			//
			IF _ResultPosition_CAL > 0 THEN 
				// calibration was completed
				// res: CAL rat:23.23 rot:23.23 err:23.23
				_VisionResult := MID(STR:=_VisionResult,LEN:=LEN(_VisionResult)-LEN(_RESPONSE_CAL),POS:=LEN(_RESPONSE_CAL)+1);
				//VisionStateText := CONCAT(VisionStateText, '\n');
				//VisionStateText := CONCAT(VisionStateText, _VisionResult);
				// rat:23.23 rot:23.23 err:23.23
				_ResultPosition := FIND(STR1:=_VisionResult,STR2:='rat:');
				IF _ResultPosition > 0 THEN
					_VisionResult := MID(STR:=_VisionResult,LEN:=LEN(_VisionResult)-LEN('rat:'),POS:=LEN('rat:')+1);
					_SpacePosition := FIND(STR1:=_VisionResult,STR2:=' ');
					_VisionRatio := STRING_TO_REAL(MID(STR:=_VisionResult,LEN:=_SpacePosition-1,POS:=1));
					_VisionResult := MID(STR:=_VisionResult,LEN:=LEN(_VisionResult)-_SpacePosition,POS:=_SpacePosition+1);
				END_IF
				// rot:23.23 err:23.23
				_ResultPosition := FIND(STR1:=_VisionResult,STR2:='rot:');
				IF _ResultPosition > 0 THEN
					_VisionResult := MID(STR:=_VisionResult,LEN:=LEN(_VisionResult)-LEN('rot:'),POS:=LEN('rot:')+1);
					_SpacePosition := FIND(STR1:=_VisionResult,STR2:=' ');
					_VisionRotation := STRING_TO_REAL(MID(STR:=_VisionResult,LEN:=_SpacePosition-1,POS:=1));
					_VisionResult := MID(STR:=_VisionResult,LEN:=LEN(_VisionResult)-_SpacePosition,POS:=_SpacePosition+1);
				END_IF
				// err:23.23
				_ResultPosition := FIND(STR1:=_VisionResult,STR2:='err:');
				IF _ResultPosition > 0 THEN
					_VisionResult := MID(STR:=_VisionResult,LEN:=LEN(_VisionResult)-LEN('err:'),POS:=LEN('err:')+1);
					_SpacePosition := FIND(STR1:=_VisionResult,STR2:=' ');
					_VisionError := STRING_TO_REAL(MID(STR:=_VisionResult,LEN:=_SpacePosition-1,POS:=1));
					_VisionResult := MID(STR:=_VisionResult,LEN:=LEN(_VisionResult)-_SpacePosition,POS:=_SpacePosition+1);
				END_IF
				
			ELSIF _ResultPosition_LOC > 0 THEN 
				// part was located
				// 'res: LOC obj:0 cx:54.66 cy:119.45 a:-12.87 s:0.84 $NLOC obj:1 cx:71.49 cy:100.06 a:10.13 s:0.83 $N'
				_VisionResult := MID(STR:=_VisionResult,LEN:=LEN(_VisionResult)-LEN(_RESPONSE_LOC),POS:=LEN(_RESPONSE_LOC)+1);
				//VisionStateText := CONCAT(VisionStateText, '\n');
				//VisionStateText := CONCAT(VisionStateText, _VisionResult);
				_VisionObjectIndex := 0;
				WHILE FIND(STR1:=_VisionResult,STR2:='obj:') > 0 
					AND _VisionObjectIndex <= _VisionCommandParser.stCommand.Locate.MaxParts 
					AND _VisionObjectIndex + _VisionCommandParser.stCommand.Locate.ResultPosition < GVL.VIS_ARR_END DO
					// 'obj:0 cx:54.66 cy:119.45 a:-12.87 s:0.84 $NLOC obj:1 cx:71.49 cy:100.06 a:10.13 s:0.83 $N'
					// $NLOC obj:1 cx:71.49 cy:100.06 a:10.13 s:0.83 $N'
					_ResultPosition := FIND(STR1:=_VisionResult,STR2:='obj:');
					IF _ResultPosition > 0 THEN
						_PartsCount := _PartsCount + 1;
						_VisionResult := MID(STR:=_VisionResult,LEN:=LEN(_VisionResult)-_ResultPosition-LEN('obj:')+1,POS:=_ResultPosition+LEN('obj:'));
						_SpacePosition := FIND(STR1:=_VisionResult,STR2:=' ');
						_VisionObjectIndex := STRING_TO_UINT(MID(STR:=_VisionResult,LEN:=_SpacePosition-1,POS:=1));
						SUPER^.VisionRegisters[_VisionCommandParser.stCommand.Locate.ResultPosition + _VisionObjectIndex].Comment := CONCAT('obj:', UDINT_TO_STRING(_VisionObjectIndex));
						_VisionResult := MID(STR:=_VisionResult,LEN:=LEN(_VisionResult)-_SpacePosition,POS:=_SpacePosition+1);
					END_IF
					// cx:54.66 cy:119.45 a:-12.87 s:0.84 $NLOC obj:1 cx:71.49 cy:100.06 a:10.13 s:0.83 $N'
					_ResultPosition := FIND(STR1:=_VisionResult,STR2:='cx:');
					IF _ResultPosition > 0 THEN
						_VisionResult := MID(STR:=_VisionResult,LEN:=LEN(_VisionResult)-LEN('cx:'),POS:=LEN('cx:')+1);
						_SpacePosition := FIND(STR1:=_VisionResult,STR2:=' ');
						SUPER^.VisionRegisters[_VisionCommandParser.stCommand.Locate.ResultPosition + _VisionObjectIndex].Position.X := STRING_TO_LREAL(MID(STR:=_VisionResult,LEN:=_SpacePosition-1,POS:=1));
						_VisionResult := MID(STR:=_VisionResult,LEN:=LEN(_VisionResult)-_SpacePosition,POS:=_SpacePosition+1);
					END_IF
					// cy:119.45 a:-12.87 s:0.84 $NLOC obj:1 cx:71.49 cy:100.06 a:10.13 s:0.83 $N'
					_ResultPosition := FIND(STR1:=_VisionResult,STR2:='cy:');
					IF _ResultPosition > 0 THEN
						_VisionResult := MID(STR:=_VisionResult,LEN:=LEN(_VisionResult)-LEN('cy:'),POS:=LEN('cy:')+1);
						_SpacePosition := FIND(STR1:=_VisionResult,STR2:=' ');
						SUPER^.VisionRegisters[_VisionCommandParser.stCommand.Locate.ResultPosition + _VisionObjectIndex].Position.Y := STRING_TO_LREAL(MID(STR:=_VisionResult,LEN:=_SpacePosition-1,POS:=1));
						_VisionResult := MID(STR:=_VisionResult,LEN:=LEN(_VisionResult)-_SpacePosition,POS:=_SpacePosition+1);
					END_IF
					// a:-12.87 s:0.84 $NLOC obj:1 cx:71.49 cy:100.06 a:10.13 s:0.83 $N'
					_ResultPosition := FIND(STR1:=_VisionResult,STR2:='a:');
					IF _ResultPosition > 0 THEN
						_VisionResult := MID(STR:=_VisionResult,LEN:=LEN(_VisionResult)-LEN('a:'),POS:=LEN('a:')+1);
						_SpacePosition := FIND(STR1:=_VisionResult,STR2:=' ');
						SUPER^.VisionRegisters[_VisionCommandParser.stCommand.Locate.ResultPosition + _VisionObjectIndex].Position.A := STRING_TO_LREAL(MID(STR:=_VisionResult,LEN:=_SpacePosition-1,POS:=1));
						_VisionResult := MID(STR:=_VisionResult,LEN:=LEN(_VisionResult)-_SpacePosition,POS:=_SpacePosition+1);
					END_IF
					// s:0.84 $NLOC obj:1 cx:71.49 cy:100.06 a:10.13 s:0.83 $N'
					_ResultPosition := FIND(STR1:=_VisionResult,STR2:='s:');
					IF _ResultPosition > 0 THEN
						_VisionResult := MID(STR:=_VisionResult,LEN:=LEN(_VisionResult)-LEN('s:'),POS:=LEN('s:')+1);
						_SpacePosition := FIND(STR1:=_VisionResult,STR2:=' ');
						SUPER^.VisionRegisters[_VisionCommandParser.stCommand.Locate.ResultPosition + _VisionObjectIndex].Scaling := STRING_TO_REAL(MID(STR:=_VisionResult,LEN:=_SpacePosition-1,POS:=1));
						_VisionResult := MID(STR:=_VisionResult,LEN:=LEN(_VisionResult)-_SpacePosition,POS:=_SpacePosition+1);
					END_IF
					// $NLOC obj:1 cx:71.49 cy:100.06 a:10.13 s:0.83 $N'
				END_WHILE
				// return how many part were found
				LogicCmdIO.Register[_VisionCommandParser.stCommand.Locate.ResultPosition] := _PartsCount;
				
			ELSIF _ResultPosition_CAP > 0 THEN 
				// image was captured
				
			END_IF
			
			//
			SUPER^._SeqMain := _STEP_DONE;
			
		END_IF

END_CASE

//
_Vision(sIpAddress:= VisionSystemIpAddress, uPort:= VisionSystemPort);

//
_VisionBusyRtrig(clk:=_Vision.P_Busy);
IF _VisionBusyRtrig.Q THEN
	VisionStateText := 'Busy';
END_IF

//
_VisionDoneRtrig(clk:=_Vision.P_Done);
IF _VisionDoneRtrig.Q THEN
	VisionStateText := 'Done';
    
    IF _ResultPosition_CAL > 0 THEN
        VisionStateText := CONCAT(VisionStateText, ': Calibration Complete');
        //VisionStateText := CONCAT(VisionStateText, _Vision.P_Response); // TODO add the response output?
        
    ELSIF _ResultPosition_LOC > 0 THEN 
        VisionStateText := CONCAT(VisionStateText, ': Found ');
        VisionStateText := CONCAT(VisionStateText, UDINT_TO_STRING(_PartsCount));
        VisionStateText := CONCAT(VisionStateText, ' parts');
        
    ELSIF _ResultPosition_CAP > 0 THEN
        VisionStateText := CONCAT(VisionStateText, ': Capture complete');
        
    END_IF
END_IF
                  

METHOD PROTECTED M_SetPackML : BOOL
                          SUPER^._UnitMode(	sName := 'Vision Processor',
				eInitialState := PACK_ML.State.Idle,
				xActive := TRUE);
                        
END_METHOD

METHOD PROTECTED M_Complete : BOOL
                          // once complete, reset to get back to idle
SUPER^._UnitMode.Reset();
                        
END_METHOD

METHOD PROTECTED M_Resetting : BOOL
                          CASE SUPER^._SeqResetting OF
	0:
		_Vision.M_Reset();
		_SeqResetting := _SeqResetting + 1;
	1:
		IF NOT _Vision.P_Error THEN
			//VisionStateText := 'RESET';
			SUPER^.M_StateComplete();
			_SeqResetting := 0;
		END_IF
END_CASE
		

                        
END_METHOD

METHOD PROTECTED M_Starting : BOOL
                          // here we want to clear things and get ready for the execute state
// I can consider this the "INIT" state
SUPER^._SeqMain := _STEP_COMMAND;
SUPER^.M_StateComplete();
                        
END_METHOD

METHOD PROTECTED M_Execute : BOOL
                          // here we want to execute our commands/jobs/etc and set completed when done.
IF SUPER^._SeqMain =_STEP_IDLE THEN
	SUPER^.M_StateComplete();
END_IF
                        
END_METHOD

METHOD PROTECTED M_Aborting : BOOL
                          CASE _SeqAborting OF
	0:
		_Vision.M_Cancel();
		_SeqAborting := _SeqAborting + 1;
		
	1: 
		IF NOT _Vision.P_Busy THEN
			SUPER^.M_StateComplete();
			_SeqAborting := 0;
		END_IF
END_CASE
                        
END_METHOD

METHOD PUBLIC M_ReconnectVisionSystem : BOOL
VAR_INPUT
END_VAR
                          // TODO may want to make sure the state machine is not in execute?
_Vision.M_Reconnect();
                        
END_METHOD

{attribute 'monitoring':='variable'}
PROPERTY PUBLIC P_PartsCount : REFERENCE TO UDINT
GET
VAR
END_VAR
                            P_PartsCount REF= _PartsCount;
                          
END_GET
END_PROPERTY

{attribute 'monitoring':='variable'}
PROPERTY PUBLIC P_VisionSystemConnected : REFERENCE TO BOOL
GET
VAR
END_VAR
                            P_VisionSystemConnected REF= _Vision._TcpClient.bConnected;
                          
END_GET
END_PROPERTY
END_FUNCTION_BLOCK

FUNCTION_BLOCK FB_ParseVarSetCmd
VAR_INPUT
	Command: STRING(GVL.COMMAND_LEN);
END_VAR
VAR_OUTPUT
	stCommand: ST_VarSetCmd;
	Error: BOOL;
	ErrorDescription: STRING;
END_VAR
VAR
	_i: INT;
	_CmdParams: ARRAY [0..GVL.COMMAND_LEN] OF STRING;
END_VAR
VAR CONSTANT
	_Delimiter: STRING:=' ';
	_ArrayTypeS: STRING(3):='STO';
	_ArrayTypeV: STRING(3):='VIS';
	_ArrayTypeF: STRING(3):='FLG';
	_OperationTypeN: STRING(1):='N';
	_OperationTypeE: STRING(1):='E';
	_OperationTypeA: STRING(1):='A';
	_OperationTypeS: STRING(1):='S';
	_OperationTypeM: STRING(1):='M';
	_OperationTypeD: STRING(1):='D';
END_VAR

                    // S|V|F index E|A|S|M|D x E|A|S|M|D yE|A|S|M|D z E|A|S|M|D a E|A|S|M|D b E|A|S|M|D c
// S 0000 E|A|S|M|D +0000.00 E|A|S|M|D +0000.00 E|A|S|M|D +0000.00 E|A|S|M|D +0000.00 E|A|S|M|D +0000.00 E|A|S|M|D +0000.00 
// V 0000 E|A|S|M|D +0000.00 E|A|S|M|D +0000.00 E|A|S|M|D +0000.00 E|A|S|M|D +0000.00 E|A|S|M|D +0000.00 E|A|S|M|D +0000.00
// F 0000 1

Error:=FALSE;
ErrorDescription:='';

// split command string into commands
_CmdParams:=F_SplitCmd(Command:=Command, _Delimiter);

//
_i:=0;
IF _CmdParams[_i] = _ArrayTypeS  THEN
	stCommand.ArrayType := DUT_Command_ArrayType.StoredPosition;
ELSIF _CmdParams[_i] = _ArrayTypeV THEN
	stCommand.ArrayType := DUT_Command_ArrayType.VisionRegister;
ELSIF _CmdParams[_i] = _ArrayTypeF THEN
	stCommand.ArrayType := DUT_Command_ArrayType.Flag;
ELSE
	Error:=TRUE;
	ErrorDescription:='Incorrect array type';
END_IF

//
_i := _i + 1;
stCommand.ArrayIndex := STRING_TO_INT(_CmdParams[_i]);
IF ((stCommand.ArrayIndex < GVL.POS_ARR_BEG OR stCommand.ArrayIndex > GVL.POS_ARR_END) AND stCommand.ArrayType = DUT_Command_ArrayType.StoredPosition)
	OR ((stCommand.ArrayIndex < GVL.VIS_ARR_BEG OR stCommand.ArrayIndex > GVL.VIS_ARR_END) AND stCommand.ArrayType = DUT_Command_ArrayType.VisionRegister)
	OR ((stCommand.ArrayIndex < GVL.FLG_ARR_BEG OR stCommand.ArrayIndex > GVL.FLG_ARR_END) AND stCommand.ArrayType = DUT_Command_ArrayType.Flag) THEN
		Error:=TRUE;
		ErrorDescription:='Incorrect array type';
END_IF

//
_i := _i + 1;
IF _CmdParams[_i] = _OperationTypeN THEN
	stCommand.XOperType := DUT_VarSetCmd_OperType.NOP;
ELSIF _CmdParams[_i] = _OperationTypeE THEN
	stCommand.XOperType := DUT_VarSetCmd_OperType.EQUALS;
ELSIF _CmdParams[_i] = _OperationTypeA THEN
	stCommand.XOperType := DUT_VarSetCmd_OperType.PLUS;
ELSIF _CmdParams[_i] = _OperationTypeS THEN
	stCommand.XOperType := DUT_VarSetCmd_OperType.MINUS;
ELSIF _CmdParams[_i] = _OperationTypeM THEN
	stCommand.XOperType := DUT_VarSetCmd_OperType.TIMES;
ELSIF _CmdParams[_i] = _OperationTypeD THEN
	stCommand.XOperType := DUT_VarSetCmd_OperType.DIVIDED_BY;
END_IF
_i := _i + 1;
stCommand.Coordinates.X := STRING_TO_LREAL(_CmdParams[_i]);

_i := _i + 1;
IF _CmdParams[_i] = _OperationTypeN THEN
	stCommand.YOperType := DUT_VarSetCmd_OperType.NOP;
ELSIF _CmdParams[_i] = _OperationTypeE THEN
	stCommand.YOperType := DUT_VarSetCmd_OperType.EQUALS;
ELSIF _CmdParams[_i] = _OperationTypeA THEN
	stCommand.YOperType := DUT_VarSetCmd_OperType.PLUS;
ELSIF _CmdParams[_i] = _OperationTypeS THEN
	stCommand.YOperType := DUT_VarSetCmd_OperType.MINUS;
ELSIF _CmdParams[_i] = _OperationTypeM THEN
	stCommand.YOperType := DUT_VarSetCmd_OperType.TIMES;
ELSIF _CmdParams[_i] = _OperationTypeD THEN
	stCommand.YOperType := DUT_VarSetCmd_OperType.DIVIDED_BY;
END_IF
_i := _i + 1;
stCommand.Coordinates.Y := STRING_TO_LREAL(_CmdParams[_i]);

_i := _i + 1;
IF _CmdParams[_i] = _OperationTypeN THEN
	stCommand.ZOperType := DUT_VarSetCmd_OperType.NOP;
ELSIF _CmdParams[_i] = _OperationTypeE THEN
	stCommand.ZOperType := DUT_VarSetCmd_OperType.EQUALS;
ELSIF _CmdParams[_i] = _OperationTypeA THEN
	stCommand.ZOperType := DUT_VarSetCmd_OperType.PLUS;
ELSIF _CmdParams[_i] = _OperationTypeS THEN
	stCommand.ZOperType := DUT_VarSetCmd_OperType.MINUS;
ELSIF _CmdParams[_i] = _OperationTypeM THEN
	stCommand.ZOperType := DUT_VarSetCmd_OperType.TIMES;
ELSIF _CmdParams[_i] = _OperationTypeD THEN
	stCommand.ZOperType := DUT_VarSetCmd_OperType.DIVIDED_BY;
END_IF
_i := _i + 1;
stCommand.Coordinates.Z := STRING_TO_LREAL(_CmdParams[_i]);

_i := _i + 1;
IF _CmdParams[_i] = _OperationTypeN THEN
	stCommand.AOperType := DUT_VarSetCmd_OperType.NOP;
ELSIF _CmdParams[_i] = _OperationTypeE THEN
	stCommand.AOperType := DUT_VarSetCmd_OperType.EQUALS;
ELSIF _CmdParams[_i] = _OperationTypeA THEN
	stCommand.AOperType := DUT_VarSetCmd_OperType.PLUS;
ELSIF _CmdParams[_i] = _OperationTypeS THEN
	stCommand.AOperType := DUT_VarSetCmd_OperType.MINUS;
ELSIF _CmdParams[_i] = _OperationTypeM THEN
	stCommand.AOperType := DUT_VarSetCmd_OperType.TIMES;
ELSIF _CmdParams[_i] = _OperationTypeD THEN
	stCommand.AOperType := DUT_VarSetCmd_OperType.DIVIDED_BY;
END_IF
_i := _i + 1;
stCommand.Coordinates.A := STRING_TO_LREAL(_CmdParams[_i]);

_i := _i + 1;
IF _CmdParams[_i] = _OperationTypeN THEN
	stCommand.BOperType := DUT_VarSetCmd_OperType.NOP;
ELSIF _CmdParams[_i] = _OperationTypeE THEN
	stCommand.BOperType := DUT_VarSetCmd_OperType.EQUALS;
ELSIF _CmdParams[_i] = _OperationTypeA THEN
	stCommand.BOperType := DUT_VarSetCmd_OperType.PLUS;
ELSIF _CmdParams[_i] = _OperationTypeS THEN
	stCommand.BOperType := DUT_VarSetCmd_OperType.MINUS;
ELSIF _CmdParams[_i] = _OperationTypeM THEN
	stCommand.BOperType := DUT_VarSetCmd_OperType.TIMES;
ELSIF _CmdParams[_i] = _OperationTypeD THEN
	stCommand.BOperType := DUT_VarSetCmd_OperType.DIVIDED_BY;
END_IF
_i := _i + 1;
stCommand.Coordinates.B := STRING_TO_LREAL(_CmdParams[_i]);

_i := _i + 1;
IF _CmdParams[_i] = _OperationTypeN THEN
	stCommand.COperType := DUT_VarSetCmd_OperType.NOP;
ELSIF _CmdParams[_i] = _OperationTypeE THEN
	stCommand.COperType := DUT_VarSetCmd_OperType.EQUALS;
ELSIF _CmdParams[_i] = _OperationTypeA THEN
	stCommand.COperType := DUT_VarSetCmd_OperType.PLUS;
ELSIF _CmdParams[_i] = _OperationTypeS THEN
	stCommand.COperType := DUT_VarSetCmd_OperType.MINUS;
ELSIF _CmdParams[_i] = _OperationTypeM THEN
	stCommand.COperType := DUT_VarSetCmd_OperType.TIMES;
ELSIF _CmdParams[_i] = _OperationTypeD THEN
	stCommand.COperType := DUT_VarSetCmd_OperType.DIVIDED_BY;
END_IF
_i := _i + 1;
stCommand.Coordinates.C := STRING_TO_LREAL(_CmdParams[_i]);
                  
END_FUNCTION_BLOCK

FUNCTION_BLOCK FB_MoveCmdProcessor EXTENDS FB_Module
VAR_INPUT
	Velocity: LREAL:=1000.0;
	VelFactor: LREAL:=1.0;
	Acceleration: LREAL:=1000.0;
	AccFactor: LREAL:=0.5;
	Jerk: LREAL:=1000.0;
	JerkFactor: LREAL:=0.5;
	Command: STRING(GVL.COMMAND_LEN):='';
END_VAR
VAR_IN_OUT
	AxisGroup: AXIS_GROUP_REF_SM3;
	GroupHandler: FB_GroupHandler;
END_VAR
VAR_OUTPUT
	Position: SMC_POS_REF;
END_VAR
VAR
	_SequenceSetCoordTrans: INT;
	_SequenceMoveCircularAbsolute: INT;
	_SequenceMoveCircularRelative: INT;
	_SequenceMoveDirectAbsolute: INT;
	_SequenceMoveDirectRelative: INT;
	_SequenceMoveLinearAbsolute: INT;
	_SequenceMoveLinearRelative: INT;
	_MC_GroupHalt: MC_GroupHalt;
	
	_MC_MoveCircularAbsolute: MC_MoveCircularAbsolute;
	_MC_MoveCircularRelative: MC_MoveCircularRelative;
	_MC_MoveDirectAbsolute: MC_MoveDirectAbsolute;
	_MC_MoveDirectRelative: MC_MoveDirectRelative;
	_MC_MoveLinearAbsolute: MC_MoveLinearAbsolute;
	_MC_MoveLinearRelative: MC_MoveLinearRelative;
	
	_UnitModeCurrentState: PACK_ML.State;
	_MoveCommandParser: FB_ParseMoveCmd;
	_PosRef: SMC_POS_REF;
	_PosRef2: SMC_POS_REF;
	
END_VAR
VAR CONSTANT
	_STEP_DONE: 				INT := 1000;
	_STEP_IDLE: 				INT := 0000;
	_STEP_COMMAND: 				INT := 0020;
	_STEP_GROUP_POWER_ON: 		INT := 0022;
	_STEP_WAIT_POWER_ON: 		INT := 0024;
	_STEP_GROUP_ENABLE: 		INT := 0030;
	_STEP_WAIT_ENABLE: 			INT := 0035;
	_STEP_READ_POSITION: 		INT := 0040;
	_STEP_WAIT_POSITION: 		INT := 0050;
	_STEP_SET_KINEMATICS: 		INT := 0060;
	_STEP_WAIT_KINEMATICS: 		INT := 0070;
	_STEP_SET_COORD_TRANS:		INT := 0071;
	_STEP_WAIT_COORD_TRANS:		INT := 0072;
	_STEP_MOVE_TYPE:			INT := 0080;
	_STEP_WAIT_MOVE: 			INT := 0090;
	_STEP_GROUP_DISABLE: 		INT := 0100;
	_STEP_WAIT_DISABLE: 		INT := 0110;
	_STEP_GROUP_POWER_OFF: 		INT := 0120;
	_STEP_ERR: 					INT := 9999;
END_VAR

                    SUPER^();

// PackML state machine implementation
_UnitModeCurrentState := SUPER^._UnitMode.CurrentState;

//
CASE SUPER^._SeqMain OF
	
	_STEP_DONE:
		SUPER^._SeqMain := _STEP_IDLE;
		
	_STEP_IDLE:
		// wait here until commanded to start
		
	_STEP_COMMAND: // parse command
		_MoveCommandParser(Command:=Command);
		SUPER^._SeqMain := _STEP_GROUP_ENABLE;
		
	_STEP_GROUP_ENABLE:
		IF GroupHandler.M_EnableGroup() THEN
			SUPER^._SeqMain := _STEP_WAIT_ENABLE;
		ELSE
			SUPER^.M_Error(Description:=CONCAT('Group Handler Error: ',
										CONCAT(TO_STRING(GroupHandler.ErrorID),
										CONCAT(' ', SMC_ErrorString(GroupHandler.ErrorID,
													SMC_Language_Type.english)))));
			SUPER^._SeqMain := _STEP_ERR; // error step so we dont spam errors
		END_IF
		
	_STEP_WAIT_ENABLE:
		// TODO add timeout timer here?
		IF GroupHandler.P_GroupEnabled THEN
			SUPER^._SeqMain := _STEP_SET_KINEMATICS;
		END_IF;
		
	_STEP_SET_KINEMATICS: // set kinematics
        // orientation convention is always ZYZ for softmotion
        GVL.OriConvention := SMC_ORI_CONVENTION.ZYZ;
        //
		_PosRef.c := _MoveCommandParser.stCommand.CoordRef;
		_PosRef2.c := _MoveCommandParser.stCommand.CoordRef2;
		IF GroupHandler.M_SetKinematics(_MoveCommandParser.stCommand.CoordSystem) THEN
			SUPER^._SeqMain := _STEP_WAIT_KINEMATICS;
		ELSE
			SUPER^.M_Error(Description:=CONCAT('Group Handler Error: ',
										CONCAT(TO_STRING(GroupHandler.ErrorID),
										CONCAT(' ', SMC_ErrorString(GroupHandler.ErrorID,
													SMC_Language_Type.english)))));
			SUPER^._SeqMain := _STEP_ERR; // error step so we dont spam errors
		END_IF
		
	_STEP_WAIT_KINEMATICS: // wait for set kinematics
		// TODO add timeout timer here?
		IF GroupHandler.P_KinematicsSet THEN
			SUPER^._SeqMain := _STEP_MOVE_TYPE;
		END_IF
		
	_STEP_MOVE_TYPE: // parse move type
		IF _MoveCommandParser.stCommand.MoveType = DUT_Command_MoveType.CircularMove THEN
			IF _MoveCommandParser.stCommand.PositionType = DUT_Command_PositionType.AbsolutePosition THEN
				_SequenceMoveCircularAbsolute := 1;
			ELSIF _MoveCommandParser.stCommand.PositionType = DUT_Command_PositionType.RelativePosition THEN
				_SequenceMoveCircularRelative := 1;
			END_IF
			
		ELSIF _MoveCommandParser.stCommand.MoveType = DUT_Command_MoveType.DirectMove THEN
			IF _MoveCommandParser.stCommand.PositionType = DUT_Command_PositionType.AbsolutePosition THEN
				_SequenceMoveDirectAbsolute := 1;
			ELSIF _MoveCommandParser.stCommand.PositionType = DUT_Command_PositionType.RelativePosition THEN
				_SequenceMoveDirectRelative := 1;
			END_IF
			
		ELSIF _MoveCommandParser.stCommand.MoveType = DUT_Command_MoveType.LinearMove THEN
			IF _MoveCommandParser.stCommand.PositionType = DUT_Command_PositionType.AbsolutePosition THEN
				_SequenceMoveLinearAbsolute := 1;
			ELSIF _MoveCommandParser.stCommand.PositionType = DUT_Command_PositionType.RelativePosition THEN
				_SequenceMoveLinearRelative := 1;
			END_IF
		END_IF
		
		SUPER^._SeqMain := _STEP_WAIT_MOVE;
		
	_STEP_WAIT_MOVE: // wait for move complete
		IF _SequenceMoveCircularAbsolute = 0
			AND _SequenceMoveCircularRelative = 0 
			AND _SequenceMoveDirectAbsolute = 0 
			AND _SequenceMoveDirectRelative = 0
			AND _SequenceMoveLinearAbsolute = 0
			AND _SequenceMoveLinearRelative = 0 THEN
				//SUPER^._SeqMain := _STEP_GROUP_DISABLE;
				SUPER^._SeqMain := _STEP_DONE;
		END_IF
	
	// TODO do we need to disable the group at this point? lets leave this here for now but skip it.
	_STEP_GROUP_DISABLE: 
		IF GroupHandler.M_DisableGroup() THEN
			SUPER^._SeqMain := _STEP_WAIT_DISABLE;
		ELSE
			SUPER^.M_Error(Description:=CONCAT('Group Handler Error: ',
										CONCAT(TO_STRING(GroupHandler.ErrorID),
										CONCAT(' ', SMC_ErrorString(GroupHandler.ErrorID,
													SMC_Language_Type.english)))));
			SUPER^._SeqMain := _STEP_ERR; // error step so we dont spam errors
		END_IF
		
	_STEP_WAIT_DISABLE:
		IF NOT GroupHandler.P_GroupEnabled THEN
			SUPER^._SeqMain := _STEP_DONE;
		END_IF
	
END_CASE

CASE _SequenceMoveCircularAbsolute OF
	0: //
	
	1: //
		_MC_MoveCircularAbsolute.Execute := TRUE;
		_SequenceMoveCircularAbsolute := 2;
		
	2: //
		IF _MC_MoveCircularAbsolute.Error THEN
			SUPER^.M_Error(Description:=CONCAT('Move Command Error: ',
										CONCAT(TO_STRING(_MC_MoveCircularAbsolute.ErrorID),
										CONCAT(' ', SMC_ErrorString(_MC_MoveCircularAbsolute.ErrorID,
													SMC_Language_Type.english)))));
			_SequenceMoveCircularAbsolute := 3; // error step so we dont spam errors
		ELSIF  _MC_MoveCircularAbsolute.Done THEN
			_MC_MoveCircularAbsolute.Execute := FALSE;
			_SequenceMoveCircularAbsolute := 0;
		END_IF
		
END_CASE

CASE _SequenceMoveCircularRelative OF
	0: //
	
	1: //
		_MC_MoveCircularRelative.Execute := TRUE;
		_SequenceMoveCircularRelative := 2;
		
	2: //
		IF _MC_MoveCircularRelative.Error THEN
			SUPER^.M_Error(Description:=CONCAT('Move Command Error: ',
										CONCAT(TO_STRING(_MC_MoveCircularRelative.ErrorID),
										CONCAT(' ', SMC_ErrorString(_MC_MoveCircularRelative.ErrorID,
													SMC_Language_Type.english)))));
			_SequenceMoveCircularRelative := 3; // error step so we dont spam errors
		ELSIF  _MC_MoveCircularRelative.Done THEN
			_MC_MoveCircularRelative.Execute := FALSE;
			_SequenceMoveCircularRelative := 0;
		END_IF
		
END_CASE

CASE _SequenceMoveDirectAbsolute OF
	0: //
	
	1: //
		_MC_MoveDirectAbsolute.Execute := TRUE;
		_SequenceMoveDirectAbsolute := 2;
		
	2: //
		IF _MC_MoveDirectAbsolute.Error THEN
			SUPER^.M_Error(Description:=CONCAT('Move Command Error: ',
										CONCAT(TO_STRING(_MC_MoveDirectAbsolute.ErrorID),
										CONCAT(' ', SMC_ErrorString(_MC_MoveDirectAbsolute.ErrorID,
													SMC_Language_Type.english)))));
			_SequenceMoveDirectAbsolute := 3; // error step so we dont spam errors
			
		ELSIF _MC_MoveDirectAbsolute.Done THEN
			_MC_MoveDirectAbsolute.Execute := FALSE;
			_SequenceMoveDirectAbsolute := 0;
		END_IF
		
END_CASE

CASE _SequenceMoveDirectRelative OF
	0: //
	
	1: //
		_MC_MoveDirectRelative.Execute := TRUE;
		_SequenceMoveDirectRelative := 2;
		
	2: //
		IF _MC_MoveDirectRelative.Error THEN
			SUPER^.M_Error(Description:=CONCAT('Move Command Error: ',
										CONCAT(TO_STRING(_MC_MoveDirectRelative.ErrorID),
										CONCAT(' ', SMC_ErrorString(_MC_MoveDirectRelative.ErrorID,
													SMC_Language_Type.english)))));
			_SequenceMoveDirectRelative := 3; // error step so we dont spam errors
			
		ELSIF _MC_MoveDirectRelative.Done THEN
			_MC_MoveDirectRelative.Execute := FALSE;
			_SequenceMoveDirectRelative := 0;
		END_IF
		
END_CASE

CASE _SequenceMoveLinearAbsolute OF
	0: //
	
	1: //
		_MC_MoveLinearAbsolute.Execute := TRUE;
		_SequenceMoveLinearAbsolute := 2;
		
	2: //
		IF _MC_MoveLinearAbsolute.Error THEN
			SUPER^.M_Error(Description:=CONCAT('Move Command Error: ',
										CONCAT(TO_STRING(_MC_MoveLinearAbsolute.ErrorID),
										CONCAT(' ', SMC_ErrorString(_MC_MoveLinearAbsolute.ErrorID,
													SMC_Language_Type.english)))));
			_SequenceMoveLinearAbsolute := 3; // error step so we dont spam errors
			
		ELSIF _MC_MoveLinearAbsolute.Done THEN
			_MC_MoveLinearAbsolute.Execute := FALSE;
			_SequenceMoveLinearAbsolute := 0;
		END_IF
END_CASE

CASE _SequenceMoveLinearRelative OF
	0: //
	
	1: //
		_MC_MoveLinearRelative.Execute := TRUE;
		_SequenceMoveLinearRelative := 2;
		
	2: //
		IF _MC_MoveLinearRelative.Error THEN
		SUPER^.M_Error(Description:=CONCAT('Move Command Error: ',
										CONCAT(TO_STRING(_MC_MoveLinearRelative.ErrorID),
										CONCAT(' ', SMC_ErrorString(_MC_MoveLinearRelative.ErrorID,
													SMC_Language_Type.english)))));
			_SequenceMoveLinearRelative := 3; // error step so we dont spam errors
			
		ELSIF _MC_MoveLinearRelative.Done THEN
			_MC_MoveLinearRelative.Execute := FALSE;
			_SequenceMoveLinearRelative := 0;
		END_IF
		
END_CASE

_MC_GroupHalt(
	AxisGroup:= AxisGroup, 
	Execute:= , 
	Deceleration:= Acceleration, 
	Jerk:= Jerk, 
	AccFactor:= AccFactor, 
	JerkFactor:= JerkFactor, 
	TorqueFactor:= , 
	ClearMovements:= , 
	Done=> , 
	Busy=> , 
	Active=> , 
	CommandAborted=> , 
	CommandAccepted=> , 
	Error=> , 
	ErrorID=> , 
	MovementId=> );

// https://content.helpme-codesys.com/de/libs/SM3_Robotics/Current/SM3_Robotics/POUs/Movement/MC_MoveCircularAbsolute.html
// https://content.helpme-codesys.com/de/libs/SM3_Robotics/Current/SM3_Robotics/Basic-types/SMC_CIRC_MODE.html#smc-circ-mode
_MC_MoveCircularAbsolute(
	AxisGroup:= AxisGroup, 
	Execute:= , 
	CircMode:= _MoveCommandParser.stCommand.CircleMode, 
	AuxPoint:= _PosRef, 
	EndPoint:= _PosRef2, 
	PathChoice:= _MoveCommandParser.stCommand.PathChoice, 
	Velocity:= Velocity, 
	Acceleration:= Acceleration, 
	Deceleration:= Acceleration, 
	Jerk:= Jerk, 
	CoordSystem:= _MoveCommandParser.stCommand.CoordSystem, 
	BufferMode:= , 
	TransitionMode:= , 
	TransitionParameter:= , 
	OrientationMode:= SMC_ORIENTATION_MODE.Axis, 
	VelFactor:= SEL(_MoveCommandParser.stCommand.Speed > 100, _MoveCommandParser.stCommand.Speed / 100.0, 1), // cannot be greater than 1
	AccFactor:= SEL(AccFactor > 1, AccFactor, 1), 
	JerkFactor:= SEL(JerkFactor > 1, JerkFactor, 1), 
	TorqueFactor:= 1, 
	Done=> , 
	Busy=> , 
	Active=> , 
	CommandAborted=> , 
	CommandAccepted=> , 
	Error=> , 
	ErrorID=> , 
	MovementId=> );

// https://content.helpme-codesys.com/en/libs/SM3_Robotics/Current/SM3_Robotics/POUs/Movement/MC_MoveCircularRelative.html
// https://content.helpme-codesys.com/de/libs/SM3_Robotics/Current/SM3_Robotics/Basic-types/SMC_CIRC_MODE.html#smc-circ-mode
_MC_MoveCircularRelative(
	AxisGroup:= AxisGroup, 
	Execute:= , 
	CircMode:= _MoveCommandParser.stCommand.CircleMode, 
	AuxPoint:= _PosRef, 
	EndPoint:= _PosRef2, 
	PathChoice:= _MoveCommandParser.stCommand.PathChoice, 
	Velocity:= Velocity, 
	Acceleration:= Acceleration, 
	Deceleration:= Acceleration, 
	Jerk:= Jerk, 
	CoordSystem:= _MoveCommandParser.stCommand.CoordSystem, 
	BufferMode:= , 
	TransitionMode:= , 
	TransitionParameter:= , 
	OrientationMode:= SMC_ORIENTATION_MODE.Axis, 
	VelFactor:= SEL(_MoveCommandParser.stCommand.Speed > 100, _MoveCommandParser.stCommand.Speed / 100.0, 1), // cannot be greater than 1
	AccFactor:= SEL(AccFactor > 1, AccFactor, 1), 
	JerkFactor:= SEL(JerkFactor > 1, JerkFactor, 1), 
	TorqueFactor:= 1, 
	Done=> , 
	Busy=> , 
	Active=> , 
	CommandAborted=> , 
	CommandAccepted=> , 
	Error=> , 
	ErrorID=> , 
	MovementId=> );
_MC_MoveDirectAbsolute(
	AxisGroup:=AxisGroup,
	Execute:= ,
	Position:= _PosRef,
	MovementType:= ,
	CoordSystem:= _MoveCommandParser.stCommand.CoordSystem,
	BufferMode:= ,
	TransitionMode:= ,
	TransitionParameter:= ,
	VelFactor:= SEL(_MoveCommandParser.stCommand.Speed > 100, _MoveCommandParser.stCommand.Speed / 100.0, 1), // cannot be greater than 1
	AccFactor:= SEL(AccFactor > 1, AccFactor, 1), 
	JerkFactor:= SEL(JerkFactor > 1, JerkFactor, 1), 
	TorqueFactor:= 1,
	Done=> ,
	Busy=> ,
	Active=> ,
	CommandAborted=> ,
	CommandAccepted=> ,
	Error=> ,
	ErrorID=> ,
	MovementId=> );
_MC_MoveDirectRelative(
	AxisGroup:= AxisGroup, 
	Execute:= , 
	Distance:= _PosRef, 
	MovementType:= , 
	CoordSystem:= _MoveCommandParser.stCommand.CoordSystem, 
	BufferMode:= , 
	TransitionMode:= , 
	TransitionParameter:= , 
	VelFactor:= SEL(_MoveCommandParser.stCommand.Speed > 100, _MoveCommandParser.stCommand.Speed / 100.0, 1), // cannot be greater than 1
	AccFactor:= SEL(AccFactor > 1, AccFactor, 1), 
	JerkFactor:= SEL(JerkFactor > 1, JerkFactor, 1), 
	TorqueFactor:= 1, 
	Done=> , 
	Busy=> , 
	Active=> , 
	CommandAborted=> , 
	CommandAccepted=> , 
	Error=> , 
	ErrorID=> , 
	MovementId=> );
	
_MC_MoveLinearAbsolute(
	AxisGroup:= AxisGroup, 
	Execute:= , 
	Position:= _PosRef,
	Velocity:= Velocity, 
	Acceleration:= Acceleration, 
	Deceleration:= Acceleration, 
	Jerk:= Jerk, 
	CoordSystem:= _MoveCommandParser.stCommand.CoordSystem, 
	BufferMode:= , 
	TransitionMode:= , 
	TransitionParameter:= , 
	OrientationMode:= SMC_ORIENTATION_MODE.Axis, 
	VelFactor:= SEL(_MoveCommandParser.stCommand.Speed > 100, _MoveCommandParser.stCommand.Speed / 100.0, 1), // cannot be greater than 1
	AccFactor:= SEL(AccFactor > 1, AccFactor, 1), 
	JerkFactor:= SEL(JerkFactor > 1, JerkFactor, 1), 
	TorqueFactor:= 1, 
	Done=> , 
	Busy=> , 
	Active=> , 
	CommandAborted=> , 
	CommandAccepted=> , 
	Error=> , 
	ErrorID=> , 
	MovementId=> );
	
_MC_MoveLinearRelative(
	AxisGroup:= AxisGroup, 
	Execute:= , 
	Distance:= _PosRef, 
	Velocity:= Velocity, 
	Acceleration:= Acceleration, 
	Deceleration:= Acceleration, 
	Jerk:= Jerk, 
	CoordSystem:= _MoveCommandParser.stCommand.CoordSystem, 
	BufferMode:= , 
	TransitionMode:= , 
	TransitionParameter:= , 
	OrientationMode:= SMC_ORIENTATION_MODE.Axis, 
	VelFactor:= SEL(_MoveCommandParser.stCommand.Speed > 100, _MoveCommandParser.stCommand.Speed / 100.0, 1), // cannot be greater than 1
	AccFactor:= SEL(AccFactor > 1, AccFactor, 1), 
	JerkFactor:= SEL(JerkFactor > 1, JerkFactor, 1), 
	TorqueFactor:= 1, 
	Done=> , 
	Busy=> , 
	Active=> , 
	CommandAborted=> , 
	CommandAccepted=> , 
	Error=> , 
	ErrorID=> , 
	MovementId=> );
                  

METHOD PROTECTED M_Starting : BOOL
                          // here we want to clear things and get ready for the execute state
// I can consider this the "INIT" state
SUPER^._SeqMain := _STEP_COMMAND;
SUPER^.M_StateComplete();
                        
END_METHOD

METHOD PROTECTED M_Resetting : BOOL
                          {warning disable C0371}
CASE SUPER^._SeqResetting OF
	0:
		GroupHandler.M_ResetGroup();
		_SeqResetting := _SeqResetting + 1;
	1:
		//IF NOT  THEN
			SUPER^.M_StateComplete();
			_SeqResetting := 0;
		//END_IF
END_CASE
{warning restore C0371}
                        
END_METHOD

METHOD PROTECTED M_Idle : BOOL
                          // in this state, we want to reset all the function blocks and hang out

_MC_MoveCircularAbsolute.Execute := FALSE;
_MC_MoveCircularRelative.Execute := FALSE;
_MC_MoveDirectAbsolute.Execute := FALSE;
_MC_MoveDirectRelative.Execute := FALSE;
_MC_MoveLinearAbsolute.Execute := FALSE;
_MC_MoveLinearRelative.Execute := FALSE;
_SequenceMoveCircularAbsolute := 0;
_SequenceMoveCircularRelative := 0;
_SequenceMoveDirectAbsolute := 0;
_SequenceMoveDirectRelative := 0;
_SequenceMoveLinearAbsolute := 0;
_SequenceMoveLinearRelative := 0;
_SequenceSetCoordTrans := 0;
SUPER^._SeqMain := 0;
                        
END_METHOD

METHOD PROTECTED M_Holding : BOOL
                          CASE SUPER^._SeqHolding OF
	0:
		_MC_MoveCircularAbsolute.Execute := FALSE;
		_MC_MoveCircularRelative.Execute := FALSE;
		_MC_MoveDirectAbsolute.Execute := FALSE;
		_MC_MoveDirectRelative.Execute := FALSE;
		_MC_MoveLinearAbsolute.Execute := FALSE;
		_MC_MoveLinearRelative.Execute := FALSE;
		_MC_GroupHalt.Execute:=TRUE;
		_SeqHolding := _SeqHolding + 1;
	1:
		IF _MC_GroupHalt.Done THEN
			_MC_GroupHalt.Execute := FALSE;
			SUPER^.M_StateComplete();
			_SeqHolding := 0;
		END_IF
		
END_CASE


                        
END_METHOD

METHOD PROTECTED M_Execute : BOOL
                          // here we want to execute our commands/jobs/etc and set completed when done.
IF SUPER^._SeqMain =_STEP_IDLE THEN
	SUPER^.M_StateComplete();
END_IF
                        
END_METHOD

METHOD PROTECTED M_Aborting : BOOL
                          {warning disable C0371}
CASE _SeqAborting OF
	0:
		GroupHandler.M_DisableGroup();
		_SeqAborting := _SeqAborting + 1;
	1:
		IF NOT GroupHandler.P_GroupEnabled THEN
			SUPER^.M_StateComplete();
			_SeqAborting := 0;
		END_IF
		
END_CASE
{warning restore C0371}
                        
END_METHOD

METHOD PROTECTED M_Complete : BOOL
                          // once complete, reset to get back to idle
SUPER^._UnitMode.Reset();
                        
END_METHOD

METHOD PROTECTED M_Unholding : BOOL
                          // here the operator called unhold (most likely from M_Start)
_MC_GroupHalt.Execute := FALSE;
CASE _MoveCommandParser.stCommand.MoveType OF 
	DUT_Command_MoveType.DirectMove:
		IF _MoveCommandParser.stCommand.PositionType = DUT_Command_Positiontype.AbsolutePosition THEN
			_MC_MoveDirectAbsolute.Execute := TRUE;
		ELSE
			_MC_MoveDirectRelative.Execute := TRUE;
		END_IF
	DUT_Command_MoveType.LinearMove:
		IF _MoveCommandParser.stCommand.PositionType = DUT_Command_Positiontype.AbsolutePosition THEN
			_MC_MoveLinearAbsolute.Execute := TRUE;
		ELSE
			_MC_MoveLinearRelative.Execute := TRUE;
		END_IF
	DUT_Command_MoveType.CircularMove:
		IF _MoveCommandParser.stCommand.PositionType = DUT_Command_Positiontype.AbsolutePosition THEN
			_MC_MoveCircularAbsolute.Execute := TRUE;
		ELSE
			_MC_MoveCircularRelative.Execute := TRUE;
		END_IF
END_CASE
//
SUPER^.M_StateComplete();
                        
END_METHOD

METHOD PROTECTED M_SetPackML : BOOL
                          SUPER^._UnitMode(	sName := 'Move Processor',
				eInitialState := PACK_ML.State.Idle,
				xActive := TRUE);
                        
END_METHOD

METHOD PROTECTED M_Clearing : BOOL
                          
_MC_MoveCircularAbsolute.Execute := FALSE;
_MC_MoveCircularRelative.Execute := FALSE;
_MC_MoveDirectAbsolute.Execute := FALSE;
_MC_MoveDirectRelative.Execute := FALSE;
_MC_MoveLinearAbsolute.Execute := FALSE;
_MC_MoveLinearRelative.Execute := FALSE;
_SequenceMoveCircularAbsolute := 0;
_SequenceMoveCircularRelative := 0;
_SequenceMoveDirectAbsolute := 0;
_SequenceMoveDirectRelative := 0;
_SequenceMoveLinearAbsolute := 0;
_SequenceMoveLinearRelative := 0;
_SequenceSetCoordTrans := 0;

SUPER^.M_StateComplete();
                        
END_METHOD
END_FUNCTION_BLOCK

FUNCTION_BLOCK FB_VarSetCmdProcessor EXTENDS FB_Module
VAR_INPUT
	Command: STRING(GVL.COMMAND_LEN):='';
END_VAR
VAR_OUTPUT
END_VAR
VAR
END_VAR
VAR CONSTANT
	_STEP_DONE: 		INT := 1000;
	_STEP_IDLE: 		INT := 0000;
	_STEP_COMMAND: 		INT := 0010;
	_STEP_ERR: 			INT := 0020;
END_VAR
VAR
	_UnitModeCurrentState: PACK_ML.State;
	_VarSetCmdParser: FB_ParseVarSetCmd;
END_VAR

                    SUPER^();

// PackML state machine implementation
_UnitModeCurrentState := SUPER^._UnitMode.CurrentState;

//
CASE SUPER^._SeqMain OF
    _STEP_DONE:
		SUPER^._SeqMain := _STEP_IDLE;
        
    _STEP_IDLE:
		// hang out here until called to run
		
	_STEP_COMMAND:
        _VarSetCmdParser(Command:=Command);
		IF _VarSetCmdParser.Error THEN
			//
			SUPER^.M_Error(Description:=_VarSetCmdParser.ErrorDescription);
			// next, please
			SUPER^._SeqMain := _STEP_ERR;
			
		ELSE
			//
			IF _VarSetCmdParser.stCommand.ArrayType = DUT_Command_ArrayType.StoredPosition THEN
				SUPER^.StoredPositions[_VarSetCmdParser.stCommand.ArrayIndex].Position.X := 
												F_VarSetCmdOperate(SUPER^.StoredPositions[_VarSetCmdParser.stCommand.ArrayIndex].Position.X, 
																	_VarSetCmdParser.stCommand.XOperType, 
																	_VarSetCmdParser.stCommand.Coordinates.X);
																	
				SUPER^.StoredPositions[_VarSetCmdParser.stCommand.ArrayIndex].Position.Y := 
												F_VarSetCmdOperate(SUPER^.StoredPositions[_VarSetCmdParser.stCommand.ArrayIndex].Position.Y, 
																	_VarSetCmdParser.stCommand.YOperType, 
																	_VarSetCmdParser.stCommand.Coordinates.Y);
																	
				SUPER^.StoredPositions[_VarSetCmdParser.stCommand.ArrayIndex].Position.Z := 
												F_VarSetCmdOperate(SUPER^.StoredPositions[_VarSetCmdParser.stCommand.ArrayIndex].Position.Z, 
																	_VarSetCmdParser.stCommand.ZOperType, 
																	_VarSetCmdParser.stCommand.Coordinates.Z);
																	
				SUPER^.StoredPositions[_VarSetCmdParser.stCommand.ArrayIndex].Position.A := 
												F_VarSetCmdOperate(SUPER^.StoredPositions[_VarSetCmdParser.stCommand.ArrayIndex].Position.A, 
																	_VarSetCmdParser.stCommand.AOperType, 
																	_VarSetCmdParser.stCommand.Coordinates.A);
																	
				SUPER^.StoredPositions[_VarSetCmdParser.stCommand.ArrayIndex].Position.B := 
												F_VarSetCmdOperate(SUPER^.StoredPositions[_VarSetCmdParser.stCommand.ArrayIndex].Position.B, 
																	_VarSetCmdParser.stCommand.BOperType, 
																	_VarSetCmdParser.stCommand.Coordinates.B);
																	
				SUPER^.StoredPositions[_VarSetCmdParser.stCommand.ArrayIndex].Position.C := 
												F_VarSetCmdOperate(SUPER^.StoredPositions[_VarSetCmdParser.stCommand.ArrayIndex].Position.C, 
																	_VarSetCmdParser.stCommand.COperType, 
																	_VarSetCmdParser.stCommand.Coordinates.C);
				
				
			ELSIF _VarSetCmdParser.stCommand.ArrayType = DUT_Command_ArrayType.VisionRegister THEN
				SUPER^.VisionRegisters[_VarSetCmdParser.stCommand.ArrayIndex].Position.X := 
												F_VarSetCmdOperate(SUPER^.VisionRegisters[_VarSetCmdParser.stCommand.ArrayIndex].Position.X, 
																	_VarSetCmdParser.stCommand.XOperType, 
																	_VarSetCmdParser.stCommand.Coordinates.X);
																	
				SUPER^.VisionRegisters[_VarSetCmdParser.stCommand.ArrayIndex].Position.Y := 
												F_VarSetCmdOperate(SUPER^.VisionRegisters[_VarSetCmdParser.stCommand.ArrayIndex].Position.Y, 
																	_VarSetCmdParser.stCommand.YOperType, 
																	_VarSetCmdParser.stCommand.Coordinates.Y);
																	
				SUPER^.VisionRegisters[_VarSetCmdParser.stCommand.ArrayIndex].Position.Z := 
												F_VarSetCmdOperate(SUPER^.VisionRegisters[_VarSetCmdParser.stCommand.ArrayIndex].Position.Z, 
																	_VarSetCmdParser.stCommand.ZOperType, 
																	_VarSetCmdParser.stCommand.Coordinates.Z);
																	
				SUPER^.VisionRegisters[_VarSetCmdParser.stCommand.ArrayIndex].Position.A := 
												F_VarSetCmdOperate(SUPER^.VisionRegisters[_VarSetCmdParser.stCommand.ArrayIndex].Position.A, 
																	_VarSetCmdParser.stCommand.AOperType, 
																	_VarSetCmdParser.stCommand.Coordinates.A);
																	
				SUPER^.VisionRegisters[_VarSetCmdParser.stCommand.ArrayIndex].Position.B := 
												F_VarSetCmdOperate(SUPER^.VisionRegisters[_VarSetCmdParser.stCommand.ArrayIndex].Position.B, 
																	_VarSetCmdParser.stCommand.BOperType, 
																	_VarSetCmdParser.stCommand.Coordinates.B);
																	
				SUPER^.VisionRegisters[_VarSetCmdParser.stCommand.ArrayIndex].Position.C := 
												F_VarSetCmdOperate(SUPER^.VisionRegisters[_VarSetCmdParser.stCommand.ArrayIndex].Position.C, 
																	_VarSetCmdParser.stCommand.COperType, 
																	_VarSetCmdParser.stCommand.Coordinates.C);
				
			ELSIF _VarSetCmdParser.stCommand.ArrayType = DUT_Command_ArrayType.Flag THEN
				// will just let the flag take on the value of X
				SUPER^.Flags[_VarSetCmdParser.stCommand.ArrayIndex].Value := LREAL_TO_BOOL(_VarSetCmdParser.stCommand.Coordinates.X);
				
			END_IF
			// next, please
			SUPER^._SeqMain := _STEP_DONE;
			
		END_IF

END_CASE
                  

METHOD PROTECTED M_SetPackML : BOOL
                          SUPER^._UnitMode(	sName := 'VarSet Processor', 
				eInitialState := PACK_ML.State.Idle,
				xActive := TRUE);
                        
END_METHOD

METHOD PROTECTED M_Complete : BOOL
                          // once complete, reset to get back to idle
SUPER^._UnitMode.Reset();
                        
END_METHOD

METHOD PROTECTED M_Starting : BOOL
                          // here we want to clear things and get ready for the execute state
// I can consider this the "INIT" state
SUPER^._SeqMain := _STEP_COMMAND;
SUPER^.M_StateComplete();
                        
END_METHOD

METHOD PROTECTED M_Execute : BOOL
                          // here we want to execute our commands/jobs/etc and set completed when done.
IF SUPER^._SeqMain =_STEP_IDLE THEN
	SUPER^.M_StateComplete();
END_IF
                        
END_METHOD
END_FUNCTION_BLOCK

FUNCTION_BLOCK FB_PauseCmdProcessor EXTENDS FB_Module
VAR_INPUT
	Command: STRING(GVL.COMMAND_LEN):='';
END_VAR
VAR_OUTPUT
	ElapsedTime: TIME;
	RemainingTime: TIME;
END_VAR
VAR
	_Timer: TON;
	_Timer_IN: BOOL;
	_Timer_PT: TIME;
	_Timer_Q: BOOL;
	_Timer_ET: TIME;
END_VAR
VAR
	_UnitModeCurrentState: PACK_ML.State;
	_ParsePauseCmd: FB_ParsePauseCmd;
END_VAR
VAR CONSTANT
	_STEP_DONE: 		INT := 1000;
	_STEP_IDLE: 		INT := 0000;
	_STEP_COMMAND: 		INT := 0010;
	_STEP_TWO: 			INT := 0020;
	_STEP_ERR: 			INT := 0030;
END_VAR

                    SUPER^();

// PackML state machine implementation
_UnitModeCurrentState := SUPER^._UnitMode.CurrentState;

//
CASE SUPER^._SeqMain OF
	
    _STEP_DONE:
 		_Timer_IN := FALSE;
		SUPER^._SeqMain := _STEP_IDLE;
        
    _STEP_IDLE:
		// hang out here until called to run
        
    _STEP_COMMAND:
		_ParsePauseCmd(Command:=Command);
		_Timer_PT := _ParsePauseCmd.stCommand.PauseTime;
 		_Timer_IN := TRUE;
		// next, please
		SUPER^._SeqMain := _STEP_TWO;
		
	_STEP_TWO:
		IF _Timer.Q THEN
			// next, please
			SUPER^._SeqMain := _STEP_DONE;
		END_IF

END_CASE

_Timer(
	IN:= _Timer_IN, 
	PT:= _Timer_PT, 
	Q=> _Timer_Q, 
	ET=> _Timer_ET);
	
ElapsedTime := _Timer_ET;
RemainingTime := _Timer_PT - _Timer_ET;
                  

METHOD PROTECTED M_SetPackML : BOOL
                          SUPER^._UnitMode(	sName := 'Pause Processor',
				eInitialState := PACK_ML.State.Idle,
				xActive := TRUE);
                        
END_METHOD

METHOD PROTECTED M_Complete : BOOL
                          // once complete, reset to get back to idle
SUPER^._UnitMode.Reset();
                        
END_METHOD

METHOD PROTECTED M_Resetting : BOOL
                          CASE SUPER^._SeqResetting OF
	0:
		_Timer_IN := FALSE;
		_SeqResetting := _SeqResetting + 1;
	1:
		IF NOT _Timer_IN THEN
			SUPER^.M_StateComplete();
			_SeqResetting := 0;
		END_IF
END_CASE
                        
END_METHOD

METHOD PROTECTED M_Execute : BOOL
                          // here we want to execute our commands/jobs/etc and set completed when done.
IF SUPER^._SeqMain =_STEP_IDLE THEN
	SUPER^.M_StateComplete();
END_IF
                        
END_METHOD

METHOD PROTECTED M_Starting : BOOL
                          // here we want to clear things and get ready for the execute state
// I can consider this the "INIT" state
SUPER^._SeqMain := _STEP_COMMAND;
SUPER^.M_StateComplete();
                        
END_METHOD
END_FUNCTION_BLOCK

FUNCTION_BLOCK FB_OutputCmdProcessor EXTENDS FB_Module
VAR_INPUT
	Enable: BOOL;
	Command: STRING(GVL.COMMAND_LEN):='';
END_VAR
VAR_IN_OUT
	Digital: ARRAY [GVL.DIG_OUT_ARR_BEG..GVL.DIG_OUT_ARR_END] OF BOOL;
	Pwm: ARRAY [GVL.PWM_OUT_ARR_BEG..GVL.PWM_OUT_ARR_END] OF BYTE;
END_VAR
VAR_OUTPUT
END_VAR
VAR
END_VAR
VAR
	_RunRtrig: R_TRIG;
	_SequenceDigital: INT;
	_SequencePwm: INT;
	
	_UnitModeCurrentState: PACK_ML.State;
	_OutputCommandParser: FB_ParseOutputCmd;
	_OutputType: DUT_OutputType;
	_OutputTarget: INT;
	_OutputValue1: LREAL;
END_VAR
VAR CONSTANT
	_STEP_DONE: 		INT := 1000;
	_STEP_IDLE: 		INT := 0000;
	_STEP_COMMAND: 		INT := 0010;
	_STEP_TWO: 			INT := 0020;
	_STEP_ERR: 			INT := 0030;
END_VAR

                    SUPER^();

// PackML state machine implementation
_UnitModeCurrentState := SUPER^._UnitMode.CurrentState;

//
CASE SUPER^._SeqMain OF
	
    _STEP_DONE:
		SUPER^._SeqMain := _STEP_IDLE;
        
    _STEP_IDLE:
        // hang out here untill called to run
		
    _STEP_COMMAND:
		_OutputCommandParser(Command:=Command);
		IF _OutputCommandParser.Error THEN
			SUPER^.M_Error(Description:=_OutputCommandParser.ErrorDescription);
			SUPER^._SeqMain := _STEP_ERR;
		ELSE
			_OutputType := _OutputCommandParser.stCommand.OutputType;
			_OutputTarget := _OutputCommandParser.stCommand.OutputTarget;
			_OutputValue1 := _OutputCommandParser.stCommand.OutputValue1;
			
			CASE _OutputType OF
				DUT_OutputType.Digital: //
					_SequenceDigital := 1;
					SUPER^._SeqMain := _STEP_TWO;
				DUT_OutputType.Pwm: //
					_SequencePwm := 1;
					SUPER^._SeqMain := _STEP_TWO;
			ELSE
				SUPER^._SeqMain := _STEP_DONE;
				
			END_CASE
		END_IF
		
	_STEP_TWO:
		IF _SequenceDigital = 0 
			AND _SequencePwm = 0 THEN
				// next, please
				SUPER^._SeqMain := _STEP_DONE;
		END_IF;

END_CASE

CASE _SequenceDigital OF
	0: //
	1: //
		THIS^.Digital[_OutputTarget] := _OutputValue1 > 0;
		_SequenceDigital := 0;
END_CASE

CASE _SequencePwm OF
	0: //
	1: //
		THIS^.Pwm[_OutputTarget] := LREAL_TO_BYTE(_OutputValue1);
		_SequencePwm := 0;
	
END_CASE
                  

METHOD PROTECTED M_SetPackML : BOOL
                          SUPER^._UnitMode(	sName := 'Output Processor',
				eInitialState := PACK_ML.State.Idle,
				xActive := TRUE);
                        
END_METHOD

METHOD PROTECTED M_Resetting : BOOL
                          CASE SUPER^._SeqResetting OF
	0:
		_SeqResetting := _SeqResetting + 1;
	1:
		SUPER^.M_StateComplete();
		_SeqResetting := 0;
END_CASE
                        
END_METHOD

METHOD PROTECTED M_Execute : BOOL
                          // here we want to execute our commands/jobs/etc and set completed when done.
IF SUPER^._SeqMain =_STEP_IDLE THEN
	SUPER^.M_StateComplete();
END_IF
                        
END_METHOD

METHOD PROTECTED M_Starting : BOOL
                          // here we want to clear things and get ready for the execute state
// I can consider this the "INIT" state
SUPER^._SeqMain := _STEP_COMMAND;
SUPER^.M_StateComplete();
                        
END_METHOD

METHOD PROTECTED M_Holding : BOOL
                          CASE SUPER^._SeqHolding OF
	0:
		SUPER^._SeqHolding := SUPER^._SeqHolding + 1;
	1:
		SUPER^.M_StateComplete();
		SUPER^._SeqHolding := 0;
		
END_CASE
                        
END_METHOD

METHOD PROTECTED M_Idle : BOOL
                          _SequenceDigital := 0;
_SequencePwm := 0;
SUPER^._SeqMain := 0;
                        
END_METHOD

METHOD PROTECTED M_Unholding : BOOL
                          
//
SUPER^._SeqMain := _STEP_COMMAND;

//
SUPER^.M_StateComplete();
                        
END_METHOD

METHOD PROTECTED M_Aborting : BOOL
                          CASE SUPER^._SeqAborting OF
	0:
		SUPER^._SeqAborting := SUPER^._SeqAborting + 1;
	1:
		SUPER^.M_StateComplete();
		SUPER^._SeqAborting := 0;
		
END_CASE

                        
END_METHOD

METHOD PROTECTED M_Clearing : BOOL
                          _SequenceDigital := 0;
_SequencePwm := 0;

SUPER^.M_StateComplete();
                        
END_METHOD

METHOD PROTECTED M_Complete : BOOL
                          // once complete, reset to get back to idle
SUPER^._UnitMode.Reset();
                        
END_METHOD
END_FUNCTION_BLOCK

{attribute 'reflection'}
FUNCTION_BLOCK FB_PackML
VAR_INPUT
END_VAR
VAR_OUTPUT
	IUnitMode: PACK_ML.IUnitMode;
END_VAR
VAR
	 {attribute 'instance-path'}
	 {attribute 'noinit'}
	 instance_path: STRING(255);
	_UnitMode: PACK_ML.UnitMode;
	_StateTimer: TON;
	_PackMLFirstScan: BOOL:=TRUE;
	_SeqMain, _SeqAborting, _SeqClearing, _SeqCompleting, _SeqHolding, _SeqResetting,
	_SeqStarting, _SeqStopping, _SeqSuspending, _SeqUnholding, _SeqUnSuspending: INT;
END_VAR
VAR CONSTANT
	STATE_TIME: TIME := T#0MS;
END_VAR

                    //
IF _PackMLFirstScan THEN
	_PackMLFirstScan := FALSE;
	M_SetPackMl();
	IUnitMode := _UnitMode;
END_IF

//
_StateTimer(PT:=STATE_TIME);

//
CASE _UnitMode.CurrentState OF
	PACK_ML.State.Stopped:
		M_Stopped();
	PACK_ML.State.Aborted:
		M_Aborted();
	PACK_ML.State.Held:
		M_Held();
	PACK_ML.State.Suspended:
		M_Suspended();
	PACK_ML.State.Complete:
		M_Complete();
	PACK_ML.State.Idle:
		M_Idle();
	PACK_ML.State.Resetting:
		M_Resetting();
	PACK_ML.State.Starting:
		M_Starting();
	PACK_ML.State.Execute:
		M_Execute();
	PACK_ML.State.Suspending:
		M_Suspending();
	PACK_ML.State.UnSuspending:
		M_UnSuspending();
	PACK_ML.State.Holding:
		M_Holding();
	PACK_ML.State.UnHolding:
		M_UnHolding();
	PACK_ML.State.Completing:
		M_Completing();
	PACK_ML.State.Aborting:
		M_Aborting();
	PACK_ML.State.Stopping:
		M_Stopping();
	PACK_ML.State.Clearing:
		M_Clearing();
END_CASE
                  

METHOD PROTECTED M_Aborting : BOOL
VAR_INPUT
END_VAR
                          _StateTimer.IN:=TRUE;

IF _StateTimer.Q THEN
	_StateTimer.IN:=FALSE;
	M_StateComplete();
END_IF
                        
END_METHOD

METHOD PROTECTED M_Unholding : BOOL
VAR_INPUT
END_VAR
                          _StateTimer.IN:=TRUE;

IF _StateTimer.Q THEN
	_StateTimer.IN:=FALSE;
	M_StateComplete();
END_IF
                        
END_METHOD

METHOD PROTECTED M_Aborted : BOOL
VAR_INPUT
END_VAR
                          _SeqMain := 0;
_SeqAborting := 0;
_SeqClearing := 0;
_SeqCompleting := 0;
_SeqHolding := 0;
_SeqResetting := 0;
_SeqStarting := 0;
_SeqStopping := 0;
_SeqSuspending := 0;
_SeqUnholding := 0;
_SeqUnSuspending := 0;
                        
END_METHOD

METHOD PROTECTED M_Held : BOOL
VAR_INPUT
END_VAR
                          (*_StateTimer.IN:=TRUE;

IF _StateTimer.Q THEN
	_StateTimer.IN:=FALSE;
	M_StateComplete();
END_IF*)
                        
END_METHOD

METHOD PROTECTED M_Completing : BOOL
VAR_INPUT
END_VAR
                          _StateTimer.IN:=TRUE;

IF _StateTimer.Q THEN
	_StateTimer.IN:=FALSE;
	M_StateComplete();
END_IF
                        
END_METHOD

METHOD PROTECTED M_Stopping : BOOL
VAR_INPUT
END_VAR
                          _StateTimer.IN:=TRUE;

IF _StateTimer.Q THEN
	_StateTimer.IN:=FALSE;
	M_StateComplete();
END_IF
                        
END_METHOD

METHOD PROTECTED M_Clearing : BOOL
VAR_INPUT
END_VAR
                          _StateTimer.IN:=TRUE;

IF _StateTimer.Q THEN
	_StateTimer.IN:=FALSE;
	M_StateComplete();
END_IF
                        
END_METHOD

METHOD PROTECTED M_Stopped : BOOL
VAR_INPUT
END_VAR
                          (*_StateTimer.IN:=TRUE;

IF _StateTimer.Q THEN
	_StateTimer.IN:=FALSE;
	M_StateComplete();
END_IF*)
                        
END_METHOD

METHOD PROTECTED M_SetPackML : BOOL
VAR_INPUT
END_VAR
                          _UnitMode(sName := 'Normal Operation', 
			dwSupportedStates := PACK_ML.State.All,
			dwAllowsLeavingFromStates := PACK_ML.State.Stopped 
											OR PACK_ML.State.Aborted 
											OR PACK_ML.State.Idle, 
			dwAllowsEnteringIntoStates := PACK_ML.State.Stopped
											OR PACK_ML.State.Aborted 
											OR PACK_ML.State.Idle, 
			eInitialState := PACK_ML.State.Idle,
			xActive := TRUE);
                        
END_METHOD

METHOD PROTECTED M_Complete : BOOL
VAR_INPUT
END_VAR
                          (*_StateTimer.IN:=TRUE;

IF _StateTimer.Q THEN
	_StateTimer.IN:=FALSE;
	M_StateComplete();
END_IF*)
                        
END_METHOD

METHOD PROTECTED M_Resetting : BOOL
VAR_INPUT
END_VAR
                          _StateTimer.IN:=TRUE;

IF _StateTimer.Q THEN
	_StateTimer.IN:=FALSE;
	M_StateComplete();
END_IF
                        
END_METHOD

METHOD PROTECTED M_Suspended : BOOL
VAR_INPUT
END_VAR
                          (*_StateTimer.IN:=TRUE;

IF _StateTimer.Q THEN
	_StateTimer.IN:=FALSE;
	M_StateComplete();
END_IF*)
                        
END_METHOD

METHOD PROTECTED M_StateComplete : BOOL
VAR_INPUT
END_VAR
                          _UnitMode.ActingStateCompleted();
                        
END_METHOD

METHOD PROTECTED M_Suspending : BOOL
VAR_INPUT
END_VAR
                          _StateTimer.IN:=TRUE;

IF _StateTimer.Q THEN
	_StateTimer.IN:=FALSE;
	M_StateComplete();
END_IF
                        
END_METHOD

METHOD PROTECTED M_Idle : BOOL
VAR_INPUT
END_VAR
                          (*_StateTimer.IN:=TRUE;

IF _StateTimer.Q THEN
	_StateTimer.IN:=FALSE;
	M_StateComplete();
END_IF*)
                        
END_METHOD

METHOD PROTECTED M_Starting : BOOL
VAR_INPUT
END_VAR
                          _StateTimer.IN:=TRUE;

IF _StateTimer.Q THEN
	_StateTimer.IN:=FALSE;
	M_StateComplete();
END_IF
                        
END_METHOD

METHOD PROTECTED M_Execute : BOOL
VAR_INPUT
END_VAR
                          
                        
END_METHOD

METHOD PROTECTED M_UnSuspending : BOOL
VAR_INPUT
END_VAR
                          _StateTimer.IN:=TRUE;

IF _StateTimer.Q THEN
	_StateTimer.IN:=FALSE;
	M_StateComplete();
END_IF
                        
END_METHOD

METHOD PROTECTED M_Holding : BOOL
VAR_INPUT
END_VAR
                          _StateTimer.IN:=TRUE;

IF _StateTimer.Q THEN
	_StateTimer.IN:=FALSE;
	M_StateComplete();
END_IF
                        
END_METHOD
END_FUNCTION_BLOCK

FUNCTION_BLOCK FB_CncCmdProcessor EXTENDS FB_Module
VAR_INPUT
	GapVelocity: LREAL := 50.0;
	AvoidGaps: BOOL := FALSE;
	GapAccel: LREAL := 100.0;
    GapJerk: LREAL := 1000.0;
	Command: STRING(GVL.COMMAND_LEN):='';
END_VAR
VAR_IN_OUT
	J1, J2, J3, J4, J5, J6: AXIS_REF_SM3;
	AxisGroup: AXIS_GROUP_REF_SM3;
	CmdIO: ST_LogicCmdIO;
END_VAR
VAR_OUTPUT
    GCodeLines: ARRAY[0..SMC_GCodeViewer.c_uiLines] OF STRING;
END_VAR
VAR
    _OriConvention: SMC_ORI_CONVENTION := SMC_ORI_CONVENTION.ZYX; // _SMC_Trafo_ArticulatedRobot_6DOF is always ZYX (yaw pitch roll) according to https://content.helpme-codesys.com/en/CODESYS%20SoftMotion/_sm_trafo_pou_six_dof_robot.html
	_SMC_TrafoConfig_ArticulatedRobot_6DOF: SMC_TrafoConfig_ArticulatedRobot_6DOF;
	_SMC_Trafo_ArticulatedRobot_6DOF: SMC_Trafo_ArticulatedRobot_6DOF;
	_SMC_ControlAxisByPos_J1: SMC_ControlAxisByPos;
	_SMC_ControlAxisByPos_J2: SMC_ControlAxisByPos;
	_SMC_ControlAxisByPos_J3: SMC_ControlAxisByPos;
	_SMC_ControlAxisByPos_J4: SMC_ControlAxisByPos;
	_SMC_ControlAxisByPos_J5: SMC_ControlAxisByPos;
	_SMC_ControlAxisByPos_J6: SMC_ControlAxisByPos;
	_SMC_Interpolator: SMC_Interpolator;
    _SMC_GCodeViewer: SMC_GCodeViewer;
    _SMC_GCODEVIEWER_DATA:  ARRAY[0..110] OF SMC_GCODEVIEWER_DATA; // must be at least interpreter queue + preprocessors
	_TrackPosition: FB_PositionTracker;
	_PlanPath: FB_CncPathPlanner;
	//_PlanPath: REFERENCE TO CncPathPlanner;
	_SysLTime, _SysLTimeLast, _CycleTime: LTIME;
    _dwCycleTime: DWORD;
	_ErrorRtrig: R_TRIG;
    _i, _j, _k: INT;
END_VAR
VAR CONSTANT
	wVarCount : WORD := 1;
    MCODE_INPUT_WAIT: INT:=200;
    MCODE_INPUT_WAIT_START: INT:=MCODE_INPUT_WAIT+GVL.DIG_IN_ARR_BEG;
    MCODE_INPUT_WAIT_END: INT:=MCODE_INPUT_WAIT+GVL.DIG_IN_ARR_END;
    MCODE_OUTPUT_SET: INT:=300;
    MCODE_OUTPUT_SET_START: INT:=MCODE_OUTPUT_SET+GVL.DIG_OUT_ARR_BEG;
    MCODE_OUTPUT_SET_END: INT:=MCODE_OUTPUT_SET+GVL.DIG_OUT_ARR_END;
    MCODE_OUTPUT_CLR: INT:=400;
    MCODE_OUTPUT_CLR_START: INT:=MCODE_OUTPUT_CLR+GVL.DIG_OUT_ARR_BEG;
    MCODE_OUTPUT_CLR_END: INT:=MCODE_OUTPUT_CLR+GVL.DIG_OUT_ARR_END;
    MCODE_FLAG_WAIT: INT:=500;
    MCODE_FLAG_WAIT_START: INT:=MCODE_FLAG_WAIT+GVL.FLG_ARR_BEG;
    MCODE_FLAG_WAIT_END: INT:=MCODE_FLAG_WAIT+GVL.FLG_ARR_END;
END_VAR
VAR CONSTANT
	_STEP_DONE: 		INT := 1000;
	_STEP_IDLE: 		INT := 0000;
	_STEP_COMMAND: 		INT := 0010;
	_STEP_ONE: 			INT := 0020;
    _STEP_ERROR:        INT := 9999;
END_VAR
VAR
	_UnitModeCurrentState: PACK_ML.State;
	_CncCmdParser: FB_ParseCncCmd;
END_VAR
VAR
	lrR1 : LREAL:=30;
	
	astVar : ARRAY [0..wVarCount] OF SMC_SingleVar :=
			[(strVarName:='R1', pAdr := ADR(lrR1), eVarType := SMC_VarType.SMC_TYPE_LREAL)];
			
	stVarList : SMC_VarList := (wNumberVars := wVarCount, psvVarlist := ADR(astVar));
END_VAR

                    // NOTE currently the settings for J6 invert direction under scaling/mapping contradict using motion control 
// libraries and CNC. For CNC to work properly, the setting is required to be enabled (inverted). Additionally
// the homing direction and position will need to be negated. This all requires a full download. Will be leaving 
// setting disabled for now so that we can continue to use motion control. 
//
// to recap, take these steps if you would like to try out CNC:
// 1. open the axis pool settings and under the scaling/mapping section enable 'invert direction'
// 2. in the A_Homing POU, change the homing direction to positive.
// 3. in _00_MAIN POU, under FirstScan set the initial home offset to a positive value (keep the value and just change the sign).
// 4. do a full download.
// 5. go online and set the persistent value (if previously initialized in FirstScan) to a positive value.
//
// UPDATE: Figured out a work around for this issue. In the A_Interpolater POU, I negated the set position in the ControlAxisByPos
// function block for J6 such that it drives the opposite way. This appears to have resolved the issue. Why this is needed, I do not
// know. I am sure it is some minor overlooked detail somewhere in the code...

// Fusion 360 Post Processor Guide: https://cam.autodesk.com/posts/posts/guides/Post%20Processor%20Training%20Guide.pdf

// path planner has to be called in a separate task with a lower priority
// https://content.helpme-codesys.com/en/libs/SM3_CNC/Current/SM_CNC_POUs/NC2/Interpreter/SMC_NCInterpreter.html
//_PlanPath REF= _60_PathPlanner.PlanPath;

SUPER^();

// PackML state machine implementation
_UnitModeCurrentState := SUPER^._UnitMode.CurrentState;

//
CASE SUPER^._SeqMain OF
    _STEP_DONE:
		_SMC_Interpolator.bExecute := FALSE;
		SUPER^._SeqMain := _STEP_IDLE;
        
    _STEP_IDLE:
		// hang out here until called to start
	
	_STEP_COMMAND:
		//
		_CncCmdParser(Command:=Command);
		_PlanPath.M_SetOriConvention(OriConvention:=_OriConvention);//_CncCmdParser.stCommand.OriConvention);
		_PlanPath.M_SetStartPosition(StartPos:=_TrackPosition.Position);//_CncCmdParser.stCommand.StartPos);
		_PlanPath.M_Execute(Filename:=_CncCmdParser.stCommand.Filename); // TODO I think we should be careful here. May need to sync CheckVelocities with the Interpolator
		
		//
		IF NOT _CncCmdParser.Error THEN
			_SMC_Interpolator.bExecute := TRUE;
			SUPER^._SeqMain := _STEP_ONE;
		ELSE
			SUPER^.M_Error(Description:=CONCAT('Command parsing error: ',_CncCmdParser.ErrorDescription));
			SUPER^._SeqMain := _STEP_ERROR;
		END_IF
        
    _STEP_ONE:
		IF NOT _SMC_Interpolator.bBusy AND NOT SUPER^.Error THEN
			// next, please
			SUPER^._SeqMain := _STEP_DONE;
		END_IF
        
    _STEP_ERROR:
        // hang out here so we dont spam errors

END_CASE

// TODO these should reference INOUT AxisGroup but somehow wont compile like that. 
// using global scoped vars for now
_SMC_TrafoConfig_ArticulatedRobot_6DOF.a1:=ArfBotAxisGroup.Trafo.a1;//AxisGroup.Trafo.a1;
_SMC_TrafoConfig_ArticulatedRobot_6DOF.a2:=ArfBotAxisGroup.Trafo.a2;//AxisGroup.Trafo.a2;
_SMC_TrafoConfig_ArticulatedRobot_6DOF.a3:=ArfBotAxisGroup.Trafo.a3;//AxisGroup.Trafo.a3;
// conflicting documentation on if d1 needs to be pos or neg. only works as negative otherwise trafo reports invalid configuration
// https://product-help.schneider-electric.com/Machine%20Expert/V2.0/zh/codesys_softmotion/codesys_softmotion/modules/_sm_trafo_pou_six_dof_robot.html
// https://forge.codesys.com/forge/talk/Motion/thread/16e1f0327f/
_SMC_TrafoConfig_ArticulatedRobot_6DOF.d1:=-ArfBotAxisGroup.Trafo.d1;//-AxisGroup.Trafo.d1;
_SMC_TrafoConfig_ArticulatedRobot_6DOF.d3:=ArfBotAxisGroup.Trafo.d3;//AxisGroup.Trafo.d3;
_SMC_TrafoConfig_ArticulatedRobot_6DOF.d4:=ArfBotAxisGroup.Trafo.d4;//AxisGroup.Trafo.d4;
_SMC_TrafoConfig_ArticulatedRobot_6DOF.d6:=ArfBotAxisGroup.Trafo.d6;//AxisGroup.Trafo.d6;
_SMC_TrafoConfig_ArticulatedRobot_6DOF.q3_max_deg:=160; // J4 // TODO put magic numbers somewhere appropriate
_SMC_TrafoConfig_ArticulatedRobot_6DOF.q3_min_deg:=-160; // J4 // TODO put magic numbers somewhere appropriate
_SMC_TrafoConfig_ArticulatedRobot_6DOF.q5_max_deg:=160; // J6 // TODO put magic numbers somewhere appropriate
_SMC_TrafoConfig_ArticulatedRobot_6DOF.q5_min_deg:=-160; // J6 // TODO put magic numbers somewhere appropriate

// TODO figure out how this var list can be used. for now its just hello world
// this gets commented out because it has to be called in a separate task with a lower priority.
_PlanPath(VarList:= stVarList, DataOut=> );

_SMC_Interpolator.bEmergency_Stop := _SMC_ControlAxisByPos_J1.bError OR _SMC_ControlAxisByPos_J1.bStopIpo
									OR _SMC_ControlAxisByPos_J2.bError OR _SMC_ControlAxisByPos_J2.bStopIpo
									OR _SMC_ControlAxisByPos_J3.bError OR _SMC_ControlAxisByPos_J3.bStopIpo
									OR _SMC_ControlAxisByPos_J4.bError OR _SMC_ControlAxisByPos_J4.bStopIpo
									OR _SMC_ControlAxisByPos_J5.bError OR _SMC_ControlAxisByPos_J5.bStopIpo
									OR _SMC_ControlAxisByPos_J6.bError OR _SMC_ControlAxisByPos_J6.bStopIpo;

// get the current measured cycle time in useconds
_SysLTime := LTIME();
_CycleTime := _SysLTime - _SysLTimeLast;
_dwCycleTime := LTIME_TO_DWORD(_CycleTime) / 1000;
_SysLTimeLast := _SysLTime;

_SMC_Interpolator(
	bExecute:= , 
	poqDataIn:= _PlanPath.DataOut, 
	bSlow_Stop:= , 
	bEmergency_Stop:= , 
	bWaitAtNextStop:= , 
	dOverride:= , 
	iVelMode:= , 
	dwIpoTime:= _dwCycleTime, //GVL.dwMainInterval,
	dLastWayPos:= , 
	bAbort:= NOT _SMC_Interpolator.bExecute, 
	bSingleStep:= , 
	bAcknM:= , 
	bQuick_Stop:= , 
	dQuickDeceleration:= , 
	dJerkMax:= , 
	dQuickStopJerk:= , 
	bSuppressSystemMFunctions:= , 
	bDone=> , 
	bBusy=> , 
	bError=> , 
	wErrorID=> , 
	piSetPosition=> , 
	iStatus=> , 
	bWorking=> , 
	iActObjectSourceNo=> , 
	dActObjectLength=> , 
	dActObjectLengthRemaining=> , 
	dVel=> , 
	vecActTangent=> , 
	iLastSwitch=> , 
	dwSwitches=> , 
	dWayPos=> , 
	wM=> , 
	adToolLength=> , 
	Act_Object=> );

// handle m codes
CASE WORD_TO_INT(_SMC_Interpolator.wM) OF
	0:	// reset acknowledgment
		_SMC_Interpolator.bAcknM := FALSE;
    
    // M200 - M215 wait on inputs 0 - 15    
	MCODE_INPUT_WAIT_START..MCODE_INPUT_WAIT_END:
        IF CmdIo.Input[WORD_TO_INT(_SMC_Interpolator.wM) - MCODE_INPUT_WAIT] THEN
            _SMC_Interpolator.bAcknM := TRUE;
        END_IF
    
    // M300 - M315 set outputs 0 - 15
	MCODE_OUTPUT_SET_START..MCODE_OUTPUT_SET_END:
        CmdIo.Output[WORD_TO_INT(_SMC_Interpolator.wM) - MCODE_OUTPUT_SET] := TRUE;
        _SMC_Interpolator.bAcknM := TRUE;
    
    // M400 - M415 clear outputs 0 - 15   
	MCODE_OUTPUT_CLR_START..MCODE_OUTPUT_CLR_END:
        CmdIo.Output[WORD_TO_INT(_SMC_Interpolator.wM) - MCODE_OUTPUT_CLR] := FALSE;
        _SMC_Interpolator.bAcknM := TRUE;
    
    // M500 - M515 wait on flags 0 - 49    
	MCODE_FLAG_WAIT_START..MCODE_FLAG_WAIT_END:
        IF SUPER^.Flags[WORD_TO_INT(_SMC_Interpolator.wM) - MCODE_FLAG_WAIT].Value THEN
            SUPER^.Flags[WORD_TO_INT(_SMC_Interpolator.wM) - MCODE_FLAG_WAIT].Value := FALSE;
            _SMC_Interpolator.bAcknM := TRUE;
        END_IF
        
END_CASE
 
_SMC_GCodeViewer(
	GCodeText:= _PlanPath.GcodeText, 
	bEnable:= _SMC_Interpolator.bBusy, 
	interpolatedObjectId:= _SMC_Interpolator.actObjectId, 
	uiNumberOfBufferEntries:=  SIZEOF(_SMC_GCODEVIEWER_DATA) / SIZEOF(SMC_GCODEVIEWER_DATA), 
	pBuffer:= ADR(_SMC_GCODEVIEWER_DATA), 
	bError=> , 
	bBusy=> , 
	wErrorID=> , 
	asGCode=> GCodeLines);

_TrackPosition(
    OriConvention:=_OriConvention,
	AxisGroup:=ArfBotAxisGroup,
	J1:=J1, J2:=J2, J3:=J3,
	J4:=J4, J5:=J5, J6:=J6,
	VisuStruct3DTrack=>,
	Arm=>,
	Elbow=>,
	Hand=>);
    
_SMC_Trafo_ArticulatedRobot_6DOF(
	config:= _SMC_TrafoConfig_ArticulatedRobot_6DOF, 
	pi:= _SMC_Interpolator.piSetPosition, 
	dQ0_old:= J1.fActPosition, 
	dQ1_old:= J2.fActPosition, 
	dQ2_old:= J3.fActPosition, 
	dQ3_old:= -J4.fActPosition,
	dQ4_old:= J5.fActPosition, 
	dQ5_old:= -J6.fActPosition, 
	armState:= _TrackPosition.Arm, 
	elbowState:= _TrackPosition.Elbow, 
	handState:= _TrackPosition.Hand, 
	dQ0=> , 
	dQ1=> , 
	dQ2=> , 
	dQ3=> , 
	dQ4=> , 
	dQ5=> , 
	bError=> , 
	result=> );
	
_SMC_ControlAxisByPos_J1(
	Axis:= J1, 
	iStatus:= _SMC_Interpolator.iStatus, 
	bEnable:= _SMC_Interpolator.bWorking, 
	bAvoidGaps:= AvoidGaps, 
	fSetPosition:= _SMC_Trafo_ArticulatedRobot_6DOF.dQ0, 
	fGapVelocity:= GapVelocity, 
	fGapAcceleration:= GapAccel, 
	fGapDeceleration:= GapAccel, 
	fGapJerk:= GapJerk, 
	bBusy=> , 
	bCommandAborted=> , 
	bError=> , 
	iErrorID=> , 
	bStopIpo=> );
	
_SMC_ControlAxisByPos_J2(
	Axis:= J2, 
	iStatus:= _SMC_Interpolator.iStatus, 
	bEnable:= _SMC_Interpolator.bWorking, 
	bAvoidGaps:= AvoidGaps, 
	fSetPosition:= _SMC_Trafo_ArticulatedRobot_6DOF.dQ1, 
	fGapVelocity:= GapVelocity, 
	fGapAcceleration:= GapAccel, 
	fGapDeceleration:= GapAccel, 
	fGapJerk:= GapJerk, 
	bBusy=> , 
	bCommandAborted=> , 
	bError=> , 
	iErrorID=> , 
	bStopIpo=> );
	
_SMC_ControlAxisByPos_J3(
	Axis:= J3, 
	iStatus:= _SMC_Interpolator.iStatus, 
	bEnable:= _SMC_Interpolator.bWorking, 
	bAvoidGaps:= AvoidGaps, 
	fSetPosition:= _SMC_Trafo_ArticulatedRobot_6DOF.dQ2, 
	fGapVelocity:= GapVelocity, 
	fGapAcceleration:= GapAccel, 
	fGapDeceleration:= GapAccel, 
	fGapJerk:= GapJerk, 
	bBusy=> , 
	bCommandAborted=> , 
	bError=> , 
	iErrorID=> , 
	bStopIpo=> );
	
_SMC_ControlAxisByPos_J4(
	Axis:= J4, 
	iStatus:= _SMC_Interpolator.iStatus, 
	bEnable:= _SMC_Interpolator.bWorking, 
	bAvoidGaps:= AvoidGaps, 
	fSetPosition:= -_SMC_Trafo_ArticulatedRobot_6DOF.dQ3,
	fGapVelocity:= GapVelocity, 
	fGapAcceleration:= GapAccel, 
	fGapDeceleration:= GapAccel, 
	fGapJerk:= GapJerk, 
	bBusy=> , 
	bCommandAborted=> , 
	bError=> , 
	iErrorID=> , 
	bStopIpo=> );
	
_SMC_ControlAxisByPos_J5(
	Axis:= J5, 
	iStatus:= _SMC_Interpolator.iStatus, 
	bEnable:= _SMC_Interpolator.bWorking, 
	bAvoidGaps:= AvoidGaps, 
	fSetPosition:= _SMC_Trafo_ArticulatedRobot_6DOF.dQ4, 
	fGapVelocity:= GapVelocity, 
	fGapAcceleration:= GapAccel, 
	fGapDeceleration:= GapAccel, 
	fGapJerk:= GapJerk, 
	bBusy=> , 
	bCommandAborted=> , 
	bError=> , 
	iErrorID=> , 
	bStopIpo=> );
	
_SMC_ControlAxisByPos_J6(
	Axis:= J6, 
	iStatus:= _SMC_Interpolator.iStatus, 
	bEnable:= _SMC_Interpolator.bWorking, 
	bAvoidGaps:= AvoidGaps, 
	fSetPosition:= -_SMC_Trafo_ArticulatedRobot_6DOF.dQ5,
	fGapVelocity:= GapVelocity, 
	fGapAcceleration:= GapAccel, 
	fGapDeceleration:= GapAccel, 
	fGapJerk:= GapJerk, 
	bBusy=> , 
	bCommandAborted=> , 
	bError=> , 
	iErrorID=> , 
	bStopIpo=> );
	
_ErrorRtrig();
_ErrorRtrig.CLK := _PlanPath.Error
					OR _SMC_Interpolator.bError
					OR _SMC_Trafo_ArticulatedRobot_6DOF.bError
					OR _SMC_ControlAxisByPos_J1.bError
					OR _SMC_ControlAxisByPos_J2.bError
					OR _SMC_ControlAxisByPos_J3.bError
					OR _SMC_ControlAxisByPos_J4.bError
					OR _SMC_ControlAxisByPos_J5.bError
					OR _SMC_ControlAxisByPos_J6.bError;
IF _ErrorRtrig.Q THEN
	IF _PlanPath.Error THEN
		SUPER^.M_Error(Description:=_PlanPath.ErrorDescription);
	END_IF
	IF _SMC_Interpolator.bError THEN
		SUPER^.M_Error(Description := CONCAT(' Interpolator Error: ',
                                CONCAT(TO_STRING(_SMC_Interpolator.wErrorID),
                                CONCAT(' ', SMC_ErrorString(_SMC_Interpolator.wErrorID,
                                            SMC_Language_Type.english)))));
	END_IF
	IF _SMC_Trafo_ArticulatedRobot_6DOF.bError THEN
		SUPER^.M_Error(Description := CONCAT(' Trafo Error: ', 'unknown'));
	END_IF
	IF _SMC_ControlAxisByPos_J1.bError THEN
        IF _SMC_ControlAxisByPos_J1.iErrorID = 183 THEN
            SUPER^.M_Error(Description := F_AxisErrorDetail(Axis := J1, AxisName := 'J1'));
        ELSE
            SUPER^.M_Error(Description :=   CONCAT(' ControlAxisByPos_J1 Error: ',
                                            CONCAT(TO_STRING(_SMC_ControlAxisByPos_J1.iErrorID),
                                            CONCAT(' ', SMC_ErrorString(_SMC_ControlAxisByPos_J1.iErrorID,
                                                    SMC_Language_Type.english)))));
        END_IF
	END_IF
	IF _SMC_ControlAxisByPos_J2.bError THEN
        IF _SMC_ControlAxisByPos_J2.iErrorID = 183 THEN
            SUPER^.M_Error(Description := F_AxisErrorDetail(Axis := J2, AxisName := 'J2'));
        ELSE
            SUPER^.M_Error(Description :=   CONCAT(' ControlAxisByPos_J2 Error: ',
                                            CONCAT(TO_STRING(_SMC_ControlAxisByPos_J2.iErrorID),
                                            CONCAT(' ', SMC_ErrorString(_SMC_ControlAxisByPos_J2.iErrorID,
                                                    SMC_Language_Type.english)))));
        END_IF
	END_IF
	IF _SMC_ControlAxisByPos_J3.bError THEN
        IF _SMC_ControlAxisByPos_J3.iErrorID = 183 THEN
            SUPER^.M_Error(Description := F_AxisErrorDetail(Axis := J3, AxisName := 'J3'));
        ELSE
            SUPER^.M_Error(Description :=   CONCAT(' ControlAxisByPos_J3 Error: ',
                                            CONCAT(TO_STRING(_SMC_ControlAxisByPos_J3.iErrorID),
                                            CONCAT(' ', SMC_ErrorString(_SMC_ControlAxisByPos_J3.iErrorID,
                                                    SMC_Language_Type.english)))));
        END_IF
	END_IF
	IF _SMC_ControlAxisByPos_J4.bError THEN
        IF _SMC_ControlAxisByPos_J4.iErrorID = 183 THEN
            SUPER^.M_Error(Description := F_AxisErrorDetail(Axis := J4, AxisName := 'J4'));
        ELSE
            SUPER^.M_Error(Description :=   CONCAT(' ControlAxisByPos_J4 Error: ',
                                            CONCAT(TO_STRING(_SMC_ControlAxisByPos_J4.iErrorID),
                                            CONCAT(' ', SMC_ErrorString(_SMC_ControlAxisByPos_J4.iErrorID,
                                                    SMC_Language_Type.english)))));
        END_IF
	END_IF
	IF _SMC_ControlAxisByPos_J5.bError THEN
        IF _SMC_ControlAxisByPos_J5.iErrorID = 183 THEN
            SUPER^.M_Error(Description := F_AxisErrorDetail(Axis := J5, AxisName := 'J5'));
        ELSE
            SUPER^.M_Error(Description :=   CONCAT(' ControlAxisByPos_J5 Error: ',
                                            CONCAT(TO_STRING(_SMC_ControlAxisByPos_J5.iErrorID),
                                            CONCAT(' ', SMC_ErrorString(_SMC_ControlAxisByPos_J5.iErrorID,
                                                    SMC_Language_Type.english)))));
        END_IF
	END_IF
	IF _SMC_ControlAxisByPos_J6.bError THEN
        IF _SMC_ControlAxisByPos_J6.iErrorID = 183 THEN
            SUPER^.M_Error(Description := F_AxisErrorDetail(Axis := J6, AxisName := 'J6'));
        ELSE
            SUPER^.M_Error(Description :=   CONCAT(' ControlAxisByPos_J6 Error: ',
                                            CONCAT(TO_STRING(_SMC_ControlAxisByPos_J6.iErrorID),
                                            CONCAT(' ', SMC_ErrorString(_SMC_ControlAxisByPos_J6.iErrorID,
                                                    SMC_Language_Type.english)))));
        END_IF
	END_IF
END_IF
                  

METHOD PROTECTED M_SetPackML : BOOL
                          SUPER^._UnitMode(	sName := 'CNC Processor',
				eInitialState := PACK_ML.State.Idle,
				xActive := TRUE);
                        
END_METHOD

METHOD PROTECTED M_Complete : BOOL
                          // once complete, reset to get back to idle
SUPER^._UnitMode.Reset();
                        
END_METHOD

METHOD PROTECTED M_Execute : BOOL
                          // here we want to execute our commands/jobs/etc and set completed when done.
IF SUPER^._SeqMain =_STEP_IDLE THEN
	SUPER^.M_StateComplete();
END_IF
                        
END_METHOD

METHOD PROTECTED M_Starting : BOOL
                          // here we want to clear things and get ready for the execute state
// I can consider this the "INIT" state
SUPER^._SeqMain := _STEP_COMMAND;
SUPER^.M_StateComplete();
                        
END_METHOD

METHOD PROTECTED M_Resetting : BOOL
                          CASE SUPER^._SeqResetting OF
	0:
		_PlanPath.M_Reset();
		_SeqResetting := _SeqResetting + 1;
	1:
		IF NOT _PlanPath.Error THEN
			SUPER^.M_StateComplete();
			_SeqResetting := 0;
		END_IF
END_CASE
                        
END_METHOD

METHOD PROTECTED M_Holding : BOOL
                          CASE _SeqHolding OF
	0:
		_SMC_Interpolator.bWaitAtNextStop := TRUE;
		SUPER^._SeqHolding := SUPER^._SeqHolding + 1;
	1:
		// TODO dale thomas this is not tested
		IF NOT _SMC_Interpolator.bWorking THEN
			SUPER^._SeqHolding := 0;
			SUPER^.M_StateComplete();
		END_IF
		
END_CASE


                        
END_METHOD

METHOD PROTECTED M_Unholding : BOOL
                          CASE _SeqUnHolding OF
	0:
		_SMC_Interpolator.bWaitAtNextStop := FALSE;
		SUPER^._SeqUnHolding := SUPER^._SeqUnHolding + 1;
	1:
		// TODO dale thomas this is not tested
		IF _SMC_Interpolator.bWorking THEN
			SUPER^._SeqUnHolding := 0;
			SUPER^.M_StateComplete();
		END_IF
		
END_CASE
                        
END_METHOD

METHOD PROTECTED M_Idle : BOOL
                          _SMC_Interpolator.bWaitAtNextStop := FALSE;
_SMC_Interpolator.bExecute := FALSE;
                        
END_METHOD
END_FUNCTION_BLOCK

FUNCTION_BLOCK FB_ParseCncCmd
VAR_INPUT
	Command: STRING(GVL.COMMAND_LEN);
END_VAR
VAR_OUTPUT
	stCommand: ST_CncCmd;
	Error: BOOL:= FALSE;
	ErrorDescription: STRING;
END_VAR
VAR
	_CmdParams: ARRAY [0..GVL.COMMAND_LEN] OF STRING;
END_VAR
VAR CONSTANT
	_AddString: STRING(3):='ADD';
	_XYZString: STRING(3):='XYZ';
	_ZYXString: STRING(3):='ZYX';
	_ZYZString: STRING(3):='ZYZ';
	_LiteralString: STRING(3):='LIT';
	_VariableString: STRING(3):='VAR';
	_StoredPositionsString: STRING(3):='STO';
	_VisionRegistersString: STRING(3):='VIS';
	_FlagsString: STRING(3):='FLG';
END_VAR

                    // /path/to/file/with/no/spaces/file.cnc ADD|XYX|ZYX|ZYZ startpos
// file1.cnc XYZ H +0250.00 +0000.00 +0500.00 +0000.00 +0045.00 +0180.00
// file2.cnc ADD A S 025
// file3.cnc ADD A V 015

// note: the command format will only contain the filename moving forward until the issues with the transformation function blocks gets resolved by CODESYS. See notes in the CncCommandProcessor about this.
// file3.cnc 

Error := FALSE;
ErrorDescription:='';

// split command string into commands
_CmdParams:=F_SplitCmd(Command:=Command);

//
IF _CmdParams[0] <> '' THEN
	//
	stCommand.Filename:=_CmdParams[0];
	
	//
	(*IF _CmdParams[1] = _AddString THEN
		stCommand.OriConvention := SMC_ORI_CONVENTION.ADDAXES;
	ELSIF _CmdParams[1] = _XYZString THEN
		stCommand.OriConvention := SMC_ORI_CONVENTION.XYZ;
	ELSIF _CmdParams[1] = _ZYXString THEN
		stCommand.OriConvention := SMC_ORI_CONVENTION.ZYX;
	ELSIF _CmdParams[1] = _ZYZString THEN
		stCommand.OriConvention := SMC_ORI_CONVENTION.ZYZ;
	ELSE
		Error := TRUE;
		ErrorDescription:='No ori convention provided';
	END_IF
	
	//
	IF _CmdParams[2] = _LiteralString THEN
		// file1.cnc XYZ H +0250.00 +0000.00 +0500.00 +0000.00 +0045.00 +0180.00
		stCommand.StartPos.dX:=STRING_TO_LREAL(_CmdParams[3]);
		stCommand.StartPos.dY:=STRING_TO_LREAL(_CmdParams[4]);
		stCommand.StartPos.dZ:=STRING_TO_LREAL(_CmdParams[5]);
		stCommand.StartPos.dA:=STRING_TO_LREAL(_CmdParams[6]);
		stCommand.StartPos.dB:=STRING_TO_LREAL(_CmdParams[7]);
		stCommand.StartPos.dC:=STRING_TO_LREAL(_CmdParams[8]);
	ELSIF _CmdParams[2] = _VariableString THEN
		// file2.cnc ADD V S 025
		IF _CmdParams[3] = _StoredPositionsString THEN
			//_ArrayType:=DUT_Command_ArrayType.StoredPosition;
			stCommand.StartPos.dX:=PersistentVars.StoredPositions[STRING_TO_INT(_CmdParams[4])].Position.X; // TODO try to remove this reference to global vars
			stCommand.StartPos.dY:=PersistentVars.StoredPositions[STRING_TO_INT(_CmdParams[4])].Position.Y;
			stCommand.StartPos.dZ:=PersistentVars.StoredPositions[STRING_TO_INT(_CmdParams[4])].Position.Z;
			stCommand.StartPos.dA:=PersistentVars.StoredPositions[STRING_TO_INT(_CmdParams[4])].Position.A;
			stCommand.StartPos.dB:=PersistentVars.StoredPositions[STRING_TO_INT(_CmdParams[4])].Position.B;
			stCommand.StartPos.dC:=PersistentVars.StoredPositions[STRING_TO_INT(_CmdParams[4])].Position.C;
		ELSIF _CmdParams[3] = _VisionRegistersString THEN
			//_ArrayType:=DUT_Command_ArrayType.Vision;
			stCommand.StartPos.dX:=PersistentVars.VisionRegisters[STRING_TO_INT(_CmdParams[4])].Position.X;
			stCommand.StartPos.dY:=PersistentVars.VisionRegisters[STRING_TO_INT(_CmdParams[4])].Position.Y;
			stCommand.StartPos.dZ:=PersistentVars.VisionRegisters[STRING_TO_INT(_CmdParams[4])].Position.Z;
			stCommand.StartPos.dA:=PersistentVars.VisionRegisters[STRING_TO_INT(_CmdParams[4])].Position.A;
			stCommand.StartPos.dB:=PersistentVars.VisionRegisters[STRING_TO_INT(_CmdParams[4])].Position.B;
			stCommand.StartPos.dC:=PersistentVars.VisionRegisters[STRING_TO_INT(_CmdParams[4])].Position.C;
		ELSIF _CmdParams[3] = _FlagsString THEN
			//_ArrayType:=DUT_Command_ArrayType.Flag;
		ELSE
			Error := TRUE;
			ErrorDescription:='No array type provided';
		END_IF
	ELSE
		Error := TRUE;
		ErrorDescription:='No variable type provided';
	END_IF*)
	
ELSE
	Error := TRUE;
	ErrorDescription:='Command string format incorrect';
	
END_IF
                  
END_FUNCTION_BLOCK

FUNCTION F_SplitCmd : ARRAY [0..GVL.COMMAND_LEN] OF STRING
VAR_INPUT
    Command: STRING(GVL.COMMAND_LEN);
	Delimiter: STRING(1):=' ';
END_VAR
VAR
	_Command: STRING(GVL.COMMAND_LEN);
	_DelimPos: INT;
	_i, _j, _k: INT;
END_VAR
VAR CONSTANT
	_SpaceChar: STRING(1):=' ';
END_VAR

                    // grab a copy
// TODO do we need to do this? cant we just operate on the input?
_Command := Command;

// ex. 123 456 789 0 123 456 879 0
WHILE LEN(_Command) > 0  AND _i < GVL.COMMAND_LEN DO
	// find the delimiter
	_DelimPos := FIND(_Command, Delimiter);
	// don't copy empty commands
	IF _DelimPos > 1 THEN
		// copy the command into the array position
		F_SplitCmd[_i] := MID(STR:=_Command, LEN:=_DelimPos - 1, POS:=1);
		// trim the command off the front of the string
		_Command := DELETE(STR:=_Command, LEN:=_DelimPos, POS:=1);
		// increment the index and get ready for the next
		_i := _i + 1;
	ELSIF _DelimPos = 1 OR FIND(_Command, _SpaceChar) = 1 THEN
		// don't do anything with a stray delimiter or a space at the  start of the next command
		// trim the command off the space at the front of the string
		_Command := DELETE(STR:=_Command, LEN:=LEN(_SpaceChar), POS:=1);
	ELSIF _DelimPos = 0 AND LEN(_Command) > 0 THEN
		// copy the last command into the array position and return
		F_SplitCmd[_i] := MID(STR:=_Command, LEN:=LEN(_Command), POS:=1);
		// trim the command off the front of the string
		_Command := DELETE(STR:=_Command, LEN:=_DelimPos, POS:=1);
		// increment the index and get ready for the next
		_i := _i + 1;
		RETURN;
	ELSE
		RETURN;
	END_IF
END_WHILE
                  
END_FUNCTION

FUNCTION F_BuildVarSetCmd : STRING(GVL.COMMAND_LEN)
VAR_INPUT
	stCommand: ST_VarSetCmd;
END_VAR
VAR
    _Command: STRING(GVL.COMMAND_LEN);
END_VAR
VAR CONSTANT
	_Delimiter: STRING:=' ';
	_ArrayTypeS: STRING(3):='STO';
	_ArrayTypeV: STRING(3):='VIS';
	_ArrayTypeF: STRING(3):='FLG';
	_OperationTypeN: STRING(1):='N';
	_OperationTypeE: STRING(1):='E';
	_OperationTypeA: STRING(1):='A';
	_OperationTypeS: STRING(1):='S';
	_OperationTypeM: STRING(1):='M';
	_OperationTypeD: STRING(1):='D';
END_VAR

                    // S|V|F index E|A|S|M|D x E|A|S|M|D yE|A|S|M|D z E|A|S|M|D a E|A|S|M|D b E|A|S|M|D c
// S 0000 E|A|S|M|D +0000.00 E|A|S|M|D +0000.00 E|A|S|M|D +0000.00 E|A|S|M|D +0000.00 E|A|S|M|D +0000.00 E|A|S|M|D +0000.00 
// V 0000 E|A|S|M|D +0000.00 E|A|S|M|D +0000.00 E|A|S|M|D +0000.00 E|A|S|M|D +0000.00 E|A|S|M|D +0000.00 E|A|S|M|D +0000.00
// F 0000 1

// clear the command
_Command:='';

// build the command
CASE stCommand.ArrayType OF
	DUT_Command_ArrayType.StoredPosition:
		F_AddElement(_Command, _Delimiter, _ArrayTypeS);
	DUT_Command_ArrayType.VisionRegister:
		F_AddElement(_Command, _Delimiter, _ArrayTypeV);
	DUT_Command_ArrayType.Flag:
		F_AddElement(_Command, _Delimiter, _ArrayTypeF);
END_CASE

// add the array index
F_AddElement(_Command, _Delimiter, INT_TO_STRING(stCommand.ArrayIndex));

// add the coordinates
IF stCommand.ArrayType = DUT_Command_ArrayType.StoredPosition 
	OR stCommand.ArrayType = DUT_Command_ArrayType.VisionRegister THEN
	
		CASE stCommand.XOperType OF
			DUT_VarSetCmd_OperType.NOP:
				F_AddElement(_Command, _Delimiter, _OperationTypeN);
			DUT_VarSetCmd_OperType.EQUALS:
				F_AddElement(_Command, _Delimiter, _OperationTypeE);
			DUT_VarSetCmd_OperType.PLUS:
				F_AddElement(_Command, _Delimiter, _OperationTypeA);
			DUT_VarSetCmd_OperType.MINUS:
				F_AddElement(_Command, _Delimiter, _OperationTypeS);
			DUT_VarSetCmd_OperType.TIMES:
				F_AddElement(_Command, _Delimiter, _OperationTypeM);
			DUT_VarSetCmd_OperType.DIVIDED_BY:
				F_AddElement(_Command, _Delimiter, _OperationTypeD);
		END_CASE
		F_AddElement(_Command, _Delimiter, LREAL_TO_STRING(stCommand.Coordinates.X));
		
		CASE stCommand.YOperType OF
			DUT_VarSetCmd_OperType.NOP:
				F_AddElement(_Command, _Delimiter, _OperationTypeN);
			DUT_VarSetCmd_OperType.EQUALS:
				F_AddElement(_Command, _Delimiter, _OperationTypeE);
			DUT_VarSetCmd_OperType.PLUS:
				F_AddElement(_Command, _Delimiter, _OperationTypeA);
			DUT_VarSetCmd_OperType.MINUS:
				F_AddElement(_Command, _Delimiter, _OperationTypeS);
			DUT_VarSetCmd_OperType.TIMES:
				F_AddElement(_Command, _Delimiter, _OperationTypeM);
			DUT_VarSetCmd_OperType.DIVIDED_BY:
				F_AddElement(_Command, _Delimiter, _OperationTypeD);
		END_CASE
		F_AddElement(_Command, _Delimiter, LREAL_TO_STRING(stCommand.Coordinates.Y));
		
		CASE stCommand.ZOperType OF
			DUT_VarSetCmd_OperType.NOP:
				F_AddElement(_Command, _Delimiter, _OperationTypeN);
			DUT_VarSetCmd_OperType.EQUALS:
				F_AddElement(_Command, _Delimiter, _OperationTypeE);
			DUT_VarSetCmd_OperType.PLUS:
				F_AddElement(_Command, _Delimiter, _OperationTypeA);
			DUT_VarSetCmd_OperType.MINUS:
				F_AddElement(_Command, _Delimiter, _OperationTypeS);
			DUT_VarSetCmd_OperType.TIMES:
				F_AddElement(_Command, _Delimiter, _OperationTypeM);
			DUT_VarSetCmd_OperType.DIVIDED_BY:
				F_AddElement(_Command, _Delimiter, _OperationTypeD);
		END_CASE;
		F_AddElement(_Command, _Delimiter, LREAL_TO_STRING(stCommand.Coordinates.Z));
		
		CASE stCommand.AOperType OF
			DUT_VarSetCmd_OperType.NOP:
				F_AddElement(_Command, _Delimiter, _OperationTypeN);
			DUT_VarSetCmd_OperType.EQUALS:
				F_AddElement(_Command, _Delimiter, _OperationTypeE);
			DUT_VarSetCmd_OperType.PLUS:
				F_AddElement(_Command, _Delimiter, _OperationTypeA);
			DUT_VarSetCmd_OperType.MINUS:
				F_AddElement(_Command, _Delimiter, _OperationTypeS);
			DUT_VarSetCmd_OperType.TIMES:
				F_AddElement(_Command, _Delimiter, _OperationTypeM);
			DUT_VarSetCmd_OperType.DIVIDED_BY:
				F_AddElement(_Command, _Delimiter, _OperationTypeD);
		END_CASE
		F_AddElement(_Command, _Delimiter, LREAL_TO_STRING(stCommand.Coordinates.A));
		
		CASE stCommand.BOperType OF
			DUT_VarSetCmd_OperType.NOP:
				F_AddElement(_Command, _Delimiter, _OperationTypeN);
			DUT_VarSetCmd_OperType.EQUALS:
				F_AddElement(_Command, _Delimiter, _OperationTypeE);
			DUT_VarSetCmd_OperType.PLUS:
				F_AddElement(_Command, _Delimiter, _OperationTypeA);
			DUT_VarSetCmd_OperType.MINUS:
				F_AddElement(_Command, _Delimiter, _OperationTypeS);
			DUT_VarSetCmd_OperType.TIMES:
				F_AddElement(_Command, _Delimiter, _OperationTypeM);
			DUT_VarSetCmd_OperType.DIVIDED_BY:
				F_AddElement(_Command, _Delimiter, _OperationTypeD);
		END_CASE
		F_AddElement(_Command, _Delimiter, LREAL_TO_STRING(stCommand.Coordinates.B));
		
		CASE stCommand.COperType OF
			DUT_VarSetCmd_OperType.NOP:
				F_AddElement(_Command, _Delimiter, _OperationTypeN);
			DUT_VarSetCmd_OperType.EQUALS:
				F_AddElement(_Command, _Delimiter, _OperationTypeE);
			DUT_VarSetCmd_OperType.PLUS:
				F_AddElement(_Command, _Delimiter, _OperationTypeA);
			DUT_VarSetCmd_OperType.MINUS:
				F_AddElement(_Command, _Delimiter, _OperationTypeS);
			DUT_VarSetCmd_OperType.TIMES:
				F_AddElement(_Command, _Delimiter, _OperationTypeM);
			DUT_VarSetCmd_OperType.DIVIDED_BY:
				F_AddElement(_Command, _Delimiter, _OperationTypeD);
		END_CASE
		F_AddElement(_Command, _Delimiter, LREAL_TO_STRING(stCommand.Coordinates.C));
		
ELSIF stCommand.ArrayType = DUT_Command_ArrayType.Flag THEN
		// we only send the x for readability. it will work if we send them all.
		F_AddElement(_Command, _Delimiter, LREAL_TO_STRING(stCommand.Coordinates.X));
		
END_IF

// set function equal to command
F_BuildVarSetCmd := _Command;
                  
END_FUNCTION

FUNCTION_BLOCK FB_LogicCmdProcessor EXTENDS FB_Module
VAR_IN_OUT
	PrgProcessor: FB_ProgramProcessor;
	CmdProcessor: FB_CommandProcessor;
	CmdIO: ST_LogicCmdIO;
END_VAR
VAR_INPUT
	Command: STRING(GVL.COMMAND_LEN):='';
END_VAR
VAR_OUTPUT
END_VAR
VAR
	_UnitModeCurrentState: PACK_ML.State;
	_ParseLogicCmd: FB_ParseLogicCmd;
	_ThenFunctionProcessed: BOOL;
END_VAR
VAR CONSTANT
	_STEP_DONE: 		INT := 1000;
	_STEP_IDLE: 		INT := 0000;
	_STEP_COMMAND: 		INT := 0010;
	_STEP_ERR: 			INT := 0020;
	_STEP_EVAL_IN:		INT := 0100;
	_STEP_EVAL_REG:		INT := 0110;
	_STEP_EVAL_CNT:		INT := 0120;
	_STEP_PROC_THEN:	INT := 0200;
	_STEP_PROC_ELSE:	INT := 0210;
	_STEP_PROC_OUT:		INT := 0300;
	_STEP_PROC_JMP:		INT := 0310;
	_STEP_PROC_CNT:		INT := 0320;
	_STEP_PROC_FLG:		INT := 0325;
	_STEP_PROC_REG:		INT := 0330;
	_STEP_EVAL_FLG:		INT := 0335;
	_STEP_PROC_NOP:		INT := 0340;
	_STEP_PROC_CAL:		INT := 0350;
END_VAR

                    SUPER^();

// PackML state machine implementation
_UnitModeCurrentState := SUPER^._UnitMode.CurrentState;

//
CASE SUPER^._SeqMain OF
	
    _STEP_DONE:
		SUPER^._SeqMain := _STEP_IDLE;
        
    _STEP_IDLE:
		// wait here until commanded to start
        
    _STEP_COMMAND:
		_ParseLogicCmd(Command:=Command);
		
		CASE _ParseLogicCmd.stCommand.IF_Condition OF
			E_LogicIfCondition.PASS:
				SUPER^._SeqMain := _STEP_PROC_THEN;
			E_LogicIfCondition.INPUT:
				SUPER^._SeqMain := _STEP_EVAL_IN;
			E_LogicIfCondition.REGISTER:
				SUPER^._SeqMain := _STEP_EVAL_REG;
			E_LogicIfCondition.COUNTER:
				SUPER^._SeqMain := _STEP_EVAL_CNT;
			E_LogicIfCondition.FLAG:
				SUPER^._SeqMain := _STEP_EVAL_FLG;
		END_CASE
		
		//
		_ThenFunctionProcessed := FALSE;
		
	_STEP_EVAL_IN:
		CASE _ParseLogicCmd.stCommand.IF_Condition_Operator OF
			E_LogicIfConditionOperator.EQU:
				IF CmdIO.Input[_ParseLogicCmd.stCommand.IF_Condition_Idx] 
					= UDINT_TO_BOOL(_ParseLogicCmd.stCommand.IF_Condition_Operator_Value) THEN
						SUPER^._SeqMain := _STEP_PROC_THEN;
				ELSE
					SUPER^._SeqMain := _STEP_PROC_ELSE;
				END_IF
			E_LogicIfConditionOperator.GRE:
				IF CmdIO.Input[_ParseLogicCmd.stCommand.IF_Condition_Idx] 
					>= UDINT_TO_BOOL(_ParseLogicCmd.stCommand.IF_Condition_Operator_Value) THEN
						SUPER^._SeqMain := _STEP_PROC_THEN;
				ELSE
					SUPER^._SeqMain := _STEP_PROC_ELSE;
				END_IF
			E_LogicIfConditionOperator.GRT:
				IF CmdIO.Input[_ParseLogicCmd.stCommand.IF_Condition_Idx] 
					> UDINT_TO_BOOL(_ParseLogicCmd.stCommand.IF_Condition_Operator_Value) THEN
						SUPER^._SeqMain := _STEP_PROC_THEN;
				ELSE
					SUPER^._SeqMain := _STEP_PROC_ELSE;
				END_IF
			E_LogicIfConditionOperator.LEQ:
				IF CmdIO.Input[_ParseLogicCmd.stCommand.IF_Condition_Idx] 
					<= UDINT_TO_BOOL(_ParseLogicCmd.stCommand.IF_Condition_Operator_Value) THEN
						SUPER^._SeqMain := _STEP_PROC_THEN;
				ELSE
					SUPER^._SeqMain := _STEP_PROC_ELSE;
				END_IF
			E_LogicIfConditionOperator.LES:
				IF CmdIO.Input[_ParseLogicCmd.stCommand.IF_Condition_Idx] 
					< UDINT_TO_BOOL(_ParseLogicCmd.stCommand.IF_Condition_Operator_Value) THEN
						SUPER^._SeqMain := _STEP_PROC_THEN;
				ELSE
					SUPER^._SeqMain := _STEP_PROC_ELSE;
				END_IF
		END_CASE
		
	_STEP_EVAL_REG:
		CASE _ParseLogicCmd.stCommand.IF_Condition_Operator OF
			E_LogicIfConditionOperator.EQU:
				IF CmdIO.Register[_ParseLogicCmd.stCommand.IF_Condition_Idx] 
					= _ParseLogicCmd.stCommand.IF_Condition_Operator_Value THEN
						SUPER^._SeqMain := _STEP_PROC_THEN;
				ELSE
					SUPER^._SeqMain := _STEP_PROC_ELSE;
				END_IF
			E_LogicIfConditionOperator.GRE:
				IF CmdIO.Register[_ParseLogicCmd.stCommand.IF_Condition_Idx] 
					>= _ParseLogicCmd.stCommand.IF_Condition_Operator_Value THEN
						SUPER^._SeqMain := _STEP_PROC_THEN;
				ELSE
					SUPER^._SeqMain := _STEP_PROC_ELSE;
				END_IF
			E_LogicIfConditionOperator.GRT:
				IF CmdIO.Register[_ParseLogicCmd.stCommand.IF_Condition_Idx] 
					> _ParseLogicCmd.stCommand.IF_Condition_Operator_Value THEN
						SUPER^._SeqMain := _STEP_PROC_THEN;
				ELSE
					SUPER^._SeqMain := _STEP_PROC_ELSE;
				END_IF
			E_LogicIfConditionOperator.LEQ:
				IF CmdIO.Register[_ParseLogicCmd.stCommand.IF_Condition_Idx] 
					<= _ParseLogicCmd.stCommand.IF_Condition_Operator_Value THEN
						SUPER^._SeqMain := _STEP_PROC_THEN;
				ELSE
					SUPER^._SeqMain := _STEP_PROC_ELSE;
				END_IF
			E_LogicIfConditionOperator.LES:
				IF CmdIO.Register[_ParseLogicCmd.stCommand.IF_Condition_Idx] 
					< _ParseLogicCmd.stCommand.IF_Condition_Operator_Value THEN
						SUPER^._SeqMain := _STEP_PROC_THEN;
				ELSE
					SUPER^._SeqMain := _STEP_PROC_ELSE;
				END_IF
		END_CASE
		
	_STEP_EVAL_CNT:
		CASE _ParseLogicCmd.stCommand.IF_Condition_Operator OF
			E_LogicIfConditionOperator.EQU:
				IF CmdIO.Counter[_ParseLogicCmd.stCommand.IF_Condition_Idx] 
					= _ParseLogicCmd.stCommand.IF_Condition_Operator_Value THEN
						SUPER^._SeqMain := _STEP_PROC_THEN;
				ELSE
					SUPER^._SeqMain := _STEP_PROC_ELSE;
				END_IF
			E_LogicIfConditionOperator.GRE:
				IF CmdIO.Counter[_ParseLogicCmd.stCommand.IF_Condition_Idx] 
					>= _ParseLogicCmd.stCommand.IF_Condition_Operator_Value THEN
						SUPER^._SeqMain := _STEP_PROC_THEN;
				ELSE
					SUPER^._SeqMain := _STEP_PROC_ELSE;
				END_IF
			E_LogicIfConditionOperator.GRT:
				IF CmdIO.Counter[_ParseLogicCmd.stCommand.IF_Condition_Idx] 
					> _ParseLogicCmd.stCommand.IF_Condition_Operator_Value THEN
						SUPER^._SeqMain := _STEP_PROC_THEN;
				ELSE
					SUPER^._SeqMain := _STEP_PROC_ELSE;
				END_IF
			E_LogicIfConditionOperator.LEQ:
				IF CmdIO.Counter[_ParseLogicCmd.stCommand.IF_Condition_Idx] 
					<= _ParseLogicCmd.stCommand.IF_Condition_Operator_Value THEN
						SUPER^._SeqMain := _STEP_PROC_THEN;
				ELSE
					SUPER^._SeqMain := _STEP_PROC_ELSE;
				END_IF
			E_LogicIfConditionOperator.LES:
				IF CmdIO.Counter[_ParseLogicCmd.stCommand.IF_Condition_Idx] 
					< _ParseLogicCmd.stCommand.IF_Condition_Operator_Value THEN
						SUPER^._SeqMain := _STEP_PROC_THEN;
				ELSE
					SUPER^._SeqMain := _STEP_PROC_ELSE;
				END_IF
		END_CASE
		
	_STEP_EVAL_FLG:
		CASE _ParseLogicCmd.stCommand.IF_Condition_Operator OF
			E_LogicIfConditionOperator.EQU:
				IF SUPER^.Flags[_ParseLogicCmd.stCommand.IF_Condition_Idx].Value 
					= UDINT_TO_BOOL(_ParseLogicCmd.stCommand.IF_Condition_Operator_Value) THEN
						SUPER^._SeqMain := _STEP_PROC_THEN;
				ELSE
					SUPER^._SeqMain := _STEP_PROC_ELSE;
				END_IF
			E_LogicIfConditionOperator.GRE:
				IF SUPER^.Flags[_ParseLogicCmd.stCommand.IF_Condition_Idx].Value  
					>= UDINT_TO_BOOL(_ParseLogicCmd.stCommand.IF_Condition_Operator_Value) THEN
						SUPER^._SeqMain := _STEP_PROC_THEN;
				ELSE
					SUPER^._SeqMain := _STEP_PROC_ELSE;
				END_IF
			E_LogicIfConditionOperator.GRT:
				IF SUPER^.Flags[_ParseLogicCmd.stCommand.IF_Condition_Idx].Value 
					> UDINT_TO_BOOL(_ParseLogicCmd.stCommand.IF_Condition_Operator_Value) THEN
						SUPER^._SeqMain := _STEP_PROC_THEN;
				ELSE
					SUPER^._SeqMain := _STEP_PROC_ELSE;
				END_IF
			E_LogicIfConditionOperator.LEQ:
				IF SUPER^.Flags[_ParseLogicCmd.stCommand.IF_Condition_Idx].Value  
					<= UDINT_TO_BOOL(_ParseLogicCmd.stCommand.IF_Condition_Operator_Value) THEN
						SUPER^._SeqMain := _STEP_PROC_THEN;
				ELSE
					SUPER^._SeqMain := _STEP_PROC_ELSE;
				END_IF
			E_LogicIfConditionOperator.LES:
				IF SUPER^.Flags[_ParseLogicCmd.stCommand.IF_Condition_Idx].Value 
					< UDINT_TO_BOOL(_ParseLogicCmd.stCommand.IF_Condition_Operator_Value) THEN
						SUPER^._SeqMain := _STEP_PROC_THEN;
				ELSE
					SUPER^._SeqMain := _STEP_PROC_ELSE;
				END_IF
		END_CASE
		
	_STEP_PROC_THEN:
		//
		_ThenFunctionProcessed := TRUE;
		//
		CASE _ParseLogicCmd.stCommand.THEN_Function OF
			E_LogicFunction.OUTPUT:
				SUPER^._SeqMain := _STEP_PROC_OUT;
			E_LogicFunction.REGISTER:
				SUPER^._SeqMain := _STEP_PROC_REG;
			E_LogicFunction.FLAG:
				SUPER^._SeqMain := _STEP_PROC_FLG;
			E_LogicFunction.CNTUP:
				SUPER^._SeqMain := _STEP_PROC_CNT;
			E_LogicFunction.CNTDN:
				SUPER^._SeqMain := _STEP_PROC_CNT;
			E_LogicFunction.CNTRST:
				SUPER^._SeqMain := _STEP_PROC_CNT;
			E_LogicFunction.JUMP:
				SUPER^._SeqMain := _STEP_PROC_JMP;
			E_LogicFunction.CALL:
				SUPER^._SeqMain := _STEP_PROC_CAL;
			E_LogicFunction.NOP:
				SUPER^._SeqMain := _STEP_PROC_NOP;
		END_CASE;
				
	_STEP_PROC_ELSE:
		IF _ParseLogicCmd.stCommand.IF_Condition <> E_LogicIfCondition.PASS THEN
			CASE _ParseLogicCmd.stCommand.ELSE_Function OF
				E_LogicFunction.OUTPUT:
					SUPER^._SeqMain := _STEP_PROC_OUT;
				E_LogicFunction.REGISTER:
					SUPER^._SeqMain := _STEP_PROC_REG;
				E_LogicFunction.FLAG:
					SUPER^._SeqMain := _STEP_PROC_FLG;
				E_LogicFunction.CNTUP:
					SUPER^._SeqMain := _STEP_PROC_CNT;
				E_LogicFunction.CNTDN:
					SUPER^._SeqMain := _STEP_PROC_CNT;
				E_LogicFunction.CNTRST:
					SUPER^._SeqMain := _STEP_PROC_CNT;
				E_LogicFunction.JUMP:
					SUPER^._SeqMain := _STEP_PROC_JMP;
				E_LogicFunction.CALL:
					SUPER^._SeqMain := _STEP_PROC_CAL;
				E_LogicFunction.NOP:
					SUPER^._SeqMain := _STEP_PROC_NOP;
			END_CASE;
		ELSE
			SUPER^._SeqMain := _STEP_DONE;
		END_IF 
		
	_STEP_PROC_OUT:
		IF _ThenFunctionProcessed THEN
			CmdIO.Output[_ParseLogicCmd.stCommand.THEN_Function_Idx] 
				:= UDINT_TO_BOOL(_ParseLogicCmd.stCommand.THEN_Function_Value);
		ELSE
			CmdIO.Output[_ParseLogicCmd.stCommand.ELSE_Function_Idx] 
				:= UDINT_TO_BOOL(_ParseLogicCmd.stCommand.ELSE_Function_Value);
		END_IF
		// next, please
		SUPER^._SeqMain := _STEP_DONE;
		
	_STEP_PROC_REG:
		IF _ThenFunctionProcessed THEN
			CmdIO.Register[_ParseLogicCmd.stCommand.THEN_Function_Idx] 
				:= _ParseLogicCmd.stCommand.THEN_Function_Value;
		ELSE
			CmdIO.Register[_ParseLogicCmd.stCommand.ELSE_Function_Idx] 
				:= _ParseLogicCmd.stCommand.ELSE_Function_Value;
		END_IF
		// next, please
		SUPER^._SeqMain := _STEP_DONE;
		
	_STEP_PROC_CNT:	
		IF _ThenFunctionProcessed THEN
			CASE _ParseLogicCmd.stCommand.THEN_Function OF
				E_LogicFunction.CNTUP:
					CmdIO.Counter[_ParseLogicCmd.stCommand.THEN_Function_Idx] 
						:= CmdIO.Counter[_ParseLogicCmd.stCommand.THEN_Function_Idx] + 1;
				E_LogicFunction.CNTDN:
					CmdIO.Counter[_ParseLogicCmd.stCommand.THEN_Function_Idx] 
						:= CmdIO.Counter[_ParseLogicCmd.stCommand.THEN_Function_Idx] - 1;
				E_LogicFunction.CNTRST:
					CmdIO.Counter[_ParseLogicCmd.stCommand.THEN_Function_Idx] 
						:= 0;
			END_CASE
		ELSE
			CASE _ParseLogicCmd.stCommand.ELSE_Function OF
				E_LogicFunction.CNTUP:
					CmdIO.Counter[_ParseLogicCmd.stCommand.ELSE_Function_Idx] 
						:= CmdIO.Counter[_ParseLogicCmd.stCommand.ELSE_Function_Idx] + 1;
				E_LogicFunction.CNTDN:
					CmdIO.Counter[_ParseLogicCmd.stCommand.ELSE_Function_Idx] 
						:= CmdIO.Counter[_ParseLogicCmd.stCommand.ELSE_Function_Idx] - 1;
				E_LogicFunction.CNTRST:
					CmdIO.Counter[_ParseLogicCmd.stCommand.ELSE_Function_Idx] 
						:= 0;
			END_CASE
		END_IF
		// next, please
		SUPER^._SeqMain := _STEP_DONE;
		
	_STEP_PROC_FLG:
		IF _ThenFunctionProcessed THEN
			SUPER^.Flags[_ParseLogicCmd.stCommand.THEN_Function_Idx].Value 
				:= UDINT_TO_BOOL(_ParseLogicCmd.stCommand.THEN_Function_Value);
		ELSE
			SUPER^.Flags[_ParseLogicCmd.stCommand.ELSE_Function_Idx].Value
				:= UDINT_TO_BOOL(_ParseLogicCmd.stCommand.ELSE_Function_Value);
		END_IF
		// next, please
		SUPER^._SeqMain := _STEP_DONE;
		
	_STEP_PROC_JMP:
		IF _ThenFunctionProcessed THEN
			CmdProcessor.M_SetNextCommand(CommandNumber:=INT_TO_UINT(_ParseLogicCmd.stCommand.THEN_Function_Idx));
		ELSE
			CmdProcessor.M_SetNextCommand(CommandNumber:=INT_TO_UINT(_ParseLogicCmd.stCommand.ELSE_Function_Idx));
		END_IF
		// next, please
		SUPER^._SeqMain := _STEP_DONE;
		
	_STEP_PROC_CAL:
		IF _ThenFunctionProcessed THEN
			PrgProcessor.M_CallProgram(	ProgramNumber:= INT_TO_UINT(_ParseLogicCmd.stCommand.THEN_Function_Idx), 
										ReturnProgram:= PrgProcessor.P_CurrentProgram, 
										ReturnCommand:= CmdProcessor.P_CurrentCommandIndex);
		ELSE
			PrgProcessor.M_CallProgram(	ProgramNumber:= INT_TO_UINT(_ParseLogicCmd.stCommand.ELSE_Function_Idx), 
										ReturnProgram:= PrgProcessor.P_CurrentProgram, 
										ReturnCommand:= CmdProcessor.P_CurrentCommandIndex);
		END_IF
		// next, please
		SUPER^._SeqMain := _STEP_DONE;
		
	_STEP_PROC_NOP:
		IF _ThenFunctionProcessed THEN
			//
		ELSE
			//
		END_IF
		// next, please
		SUPER^._SeqMain := _STEP_DONE;

END_CASE
                  

METHOD PROTECTED M_SetPackML : BOOL
                          SUPER^._UnitMode(	sName := 'Logic Processor',
				eInitialState := PACK_ML.State.Idle,
				xActive := TRUE);
                        
END_METHOD

METHOD PROTECTED M_Complete : BOOL
                          // once complete, reset to get back to idle
SUPER^._UnitMode.Reset();
                        
END_METHOD

METHOD PROTECTED M_Execute : BOOL
                          // here we want to execute our commands/jobs/etc and set completed when done.
IF SUPER^._SeqMain =_STEP_IDLE THEN
	SUPER^.M_StateComplete();
END_IF
                        
END_METHOD

METHOD PROTECTED M_Starting : BOOL
                          // here we want to clear things and get ready for the execute state
// I can consider this the "INIT" state
SUPER^._SeqMain := _STEP_COMMAND;
SUPER^.M_StateComplete();
                        
END_METHOD
END_FUNCTION_BLOCK

FUNCTION F_AddElement
VAR_IN_OUT
	Command: STRING(GVL.COMMAND_LEN);
END_VAR
VAR_INPUT
	Delimiter: STRING(1):=' '; // default to space
	Element: STRING(GVL.COMMAND_LEN);
END_VAR
VAR
END_VAR

                    //
// input
// 	Element: 'bar'
// 	Delimiter: ','
// 	Command: 'foo'
//
// output
// 	Command: 'foo,bar'
//

Command:=CONCAT(Command, Element);
Command:=CONCAT(Command, Delimiter);
                  
END_FUNCTION

FUNCTION F_BuildMoveCmd : STRING(GVL.COMMAND_LEN);
VAR_INPUT
	stCommand: ST_MoveCmd;
END_VAR
VAR
	_Command : STRING(GVL.COMMAND_LEN);
END_VAR
VAR CONSTANT
	_Delimiter: STRING:=' ';
	_MoveTypeD: STRING(3):='DIR';
	_MoveTypeL: STRING(3):='LIN';
	_MoveTypeC: STRING(3):='CIR';
	_ChangeTypeA: STRING(3):='ABS';
	_ChangeTypeR: STRING(3):='REL';
	_CoordSystemAcs: STRING(3):='ACS';
	_CoordSystemMcs: STRING(3):='MCS';
	_CoordSystemPc1: STRING(3):='PC1';
	_CoordSystemPc2: STRING(3):='PC2';
	_CoordSystemTcs: STRING(3):='TCS';
	_CoordSystemWcs: STRING(3):='WCS';
	_CoordSystemIcs: STRING(3):='ICS';
	_CoordTypeH: STRING(3):='LIT';
	_CoordTypeV: STRING(3):='VAR';
	_ArrayTypeS: STRING(3):='STO';
	_ArrayTypeV: STRING(3):='VIS';
	_ArrayTypeF: STRING(3):='FLG';
	_CircleModeBor: STRING(3):='BOR';
	_CircleModeCen: STRING(3):='CEN';
	_CircleModeRad: STRING(3):='RAD';
	_PathChoiceClw: STRING(3):='CLW';
	_PathChoiceCcw: STRING(3):='CCW';
END_VAR

                    // D is direct move. L is linear move. C is a circular move
// R is relative position. A is absolute position
// V is variable coordinated. H is a hardcoded coordinated
// S is stored position array. V is vision register array.
// D|L|C R|A Speed CoordSystem X0000.00 Y0000.00 Z0000.00 A0000.00 B0000.00 C0000.00 BOR|CEN|RAD CCW|CLW X0000.00 Y0000.00 Z0000.00 A0000.00 B0000.00 C0000.00
// 'D A 010 MCS H +0250.00 +0000.00 +0500.00 +0000.00 +0045.00 +0180.00'
// 'C R 010 MCS H +0250.00 +0000.00 +0500.00 +0000.00 +0045.00 +0180.00 BOR CLW H +0250.00 +0000.00 +0500.00 +0000.00 +0045.00 +0180.00'
// 'D A 010 MCS V S 025'
// 'D A 010 MCS V V 033'
// 'C R 010 MCS V S 002 BOR CLW V S 005'
// 'C R 010 MCS V S 003 BOR CLW V V 006'
// 'C R 010 MCS V S 015 BOR CLW H +0250.00 +0000.00 +0500.00 +0000.00 +0045.00 +0180.00'
// 'C R 010 MCS H +0250.00 +0000.00 +0500.00 +0000.00 +0045.00 +0180.00 BOR CLW V V 022'

//
_Command := '';

//
CASE stCommand.MoveType OF
	DUT_Command_MoveType.DirectMove:
		F_AddElement(_Command, _Delimiter, _MoveTypeD);
	DUT_Command_MoveType.LinearMove:
		F_AddElement(_Command, _Delimiter, _MoveTypeL);
	DUT_Command_MoveType.CircularMove:
		F_AddElement(_Command, _Delimiter, _MoveTypeC);
END_CASE

